FUNCTION "FC20 Motor 1O1I" : VOID	// FC 20
TITLE = Block for motor actuation and fault monitoring
//Erstellung:
//Datum        Bearbeiter                                                 Version
//--------------------------------------------------------------------------------
//26.06.97     H.Rüttling (rh)                                            01.00.00
//
//Änderungen:
//Nr. Datum    Bearb Änderung                                       Marke  Version
//--------------------------------------------------------------------------------
//01  09.02.99 sra   Einfügen der Handbedienuung                    ()    01.01.00
//02  16.04.99 sra   Fehlerbeseitigung Störungsquittierung          ()    01.01.01
//03  23.07.99 sra   Ausg. wird auch bei Simulation gesetzt         ()    01.01.02
//04  19.10.99 sra   "in" Reparaturschalter gelöscht                ()    01.02.00
//05  03.11.99 hus   Parameter eingefügt "FU in Betrieb"            ()    01.03.00
//06  18.09.00 sra   komplette Überarbeitung / neue Struktur        ()    02.00.00
//07  08.11.02 sra   Änderung Betriebsstundenzähler (zählt falsch)  (007) 02.01.00
//08  31.10.05 sra   Ansteuerung Handbedienung im Automode rücksetz.
//                   Handbedienung zentral sperren                  (008) 02.02.00
//09  04.09.06 sra   Änderung Störungsquittierung                   (009) 02.03.00
//10  20.11.07 gea   Handmode zurücksetzen wenn Handmode gesperrt   (010) 02.03.01
//11  18.02.09 kmj   Objektststatus für OP ergänzt                  (011) 02.04.00
//12  20.03.09 kal   Objektststatus für OP ergänzt (überarbeitet)   (012) 02.04.01
//13  05.12.13 sra   "Anlage ein" eingefügt (Not-Aus-Konzept)       (013) 02.05.00
//________________________________________________________________________________
//Funktion:
//
//-Der Baustein steuert den Ablauf eines Motors mit 1 Ausgang und 1 Eingang durch 
// setzten des Eingangsparameters "in_Ansteuerung_Motor".
//
//-Der Ausgang wird nur angesteuert wenn der Eingang "in_Anlage_ein" = true
// ist. Diese Funktion ist vorhanden, um bei einem Not-Halt die Anlage vor 
// unkontrolliertem Einschalten zu schützen. 
//
//-Ist in der Motorstruktur die Taktfunktion freigegeben wird bei Freigabe des 
// Motors der Ausgang entsprechend der Impuls-/Pausezeit angesteuert.
// !!Der Baustein arbeitet nur mit vollen Sekunden!!
//
//-Der Baustein überwacht den Zustand des Ausgangs und des Eingangs und generiert 
// nach Ablauf der "Sollzeit Störung" eine Störmeldung
//
//-Ist das Bit "Simulation" auf TRUE, so wird der Eingang simuliert.
//
//-Ist die Kennung "Betriebsstundenzähler_ein" aktiviert werden die Laufzeit 
// des Motors aufsummiert. Dies erfolgt mit setzen des Ausgangs.
//
//-Der Baustein kopiert die Parameter "in_Eingang_Motor", "io_Ausgang_Motor", 
// "in_Quitt_Stoerung" und "io_Stoerung" in die angegebene Datenstruktur zur 
// Visualisierung auf einem Farbgrafiksystem. Diese Parameter müssen folglich 
// nicht mehr extern umkopiert werden.
//
//-Ist der Parameter "in_Handbedienung_erlaubt" angewählt kann der Motor über 
// eine Farbgrafik oder ein Bedienterminal manuell angesteuert werden
//
AUTHOR : rh
FAMILY : AZO
VERSION : 0.0
VAR_INPUT
  in_Handbedienung_erlaubt : BOOL ;	//1 = manual operation permitted, 0 = manual operation not permitted/locked
  in_Quitt_Stoerung_noetig : BOOL ;	//1 = fault acknowledgement required, 0 = automatic fault acknowledgement
  in_Anlage_ein : BOOL ;	//Anlage bzw. Anlagenbereich nach Not-Halt freigegeben
  in_Quitt_Stoerung : BOOL ;	//Fault acknowledgement when fault_acknowledgement_required = 1
  in_Ansteuerung_Motor : BOOL ;	//Actuation of motor in automatic mode
  in_Eingang_Motor : BOOL ;	//Input of motor
END_VAR
VAR_IN_OUT
  io_Ausgang_Motor : BOOL ;	//Output of motor
  io_Motor_in_Betrieb : BOOL ;	//Signal "motor in operation"
  io_Stoerung : BOOL ;	//Signal "motor fault"
  io_Motorstruktur : ANY ;	//ANY pointer of motor structure
END_VAR
VAR_TEMP
  Freigabe_Takt : BOOL ;
  Start_mit_Impuls : BOOL ;
  Dauertakt : BOOL ;
  Taktausgang : BOOL ;
  Taktanzahl_erreicht : BOOL ;
  Diskrepanz : BOOL ;
  Impulszeit : REAL ;
  Pausezeit : REAL ;
  Sollanzahl_Takte : INT ;
  Zeitzaehler : REAL ;
  Taktzaehler : INT ;
  Objektstatus : INT ;
END_VAR
BEGIN
NETWORK
TITLE = Anfangs-DW der Struktur aus ANY-Zeiger auslesen
      L     P##io_Motorstruktur;
      LAR2;
      L     D [AR2,P#6.0];
      LAR2;
NETWORK
TITLE = Simulation
      AN    DIX [AR2,P#3.5];	// Simulation ein (Struktur)
      JC    ESIM;
      A     #io_Ausgang_Motor;
      =     #in_Eingang_Motor;
ESIM: NOP   0;
NETWORK
TITLE = Umschaltung Hand-/Automatikmode 
      A     DIX [AR2,P#2.7];	// Handmode von Farbgrafik (Struktur)
      AN    DIX [AR2,P#3.1];	// Handmode gesperrt (Struktur)
      AN    "M 0.0 Lock Man.Operation";	// Handbedienung zentral sperren (008)
      S     DIX [AR2,P#2.6];	// Handmode zu Farbgrafik (Struktur)
      ON    DIX [AR2,P#2.7];	// Handmode von Farbgrafik (Struktur)
      ON    #in_Handbedienung_erlaubt;
      O     "M 0.0 Lock Man.Operation";	// Handbedienung zentral sperren (008)
      O     DIX [AR2,P#3.1];	// Handmode gesperrt (Struktur)//(010)
      R     DIX [AR2,P#2.6];	// Handmode zu Farbgrafik (Struktur)
      R     DIX [AR2,P#2.7];	// Handmode zu Farbgrafik (Struktur) (008)
NETWORK
TITLE = Ansteuerung Handmode zurücksetzen
//(008) 
      AN    DIX [AR2,P#2.6];	// Handmode zu Farbgrafik (Struktur)
      R     DIX [AR2,P#3.0];	// Ansteuerung Handmode von Farbgrafik (Struktur)
NETWORK
TITLE = Daten für Takt in temporäre Variablen laden
      A     #in_Anlage_ein;	// (013)
      A     #in_Ansteuerung_Motor;
      A     DIX [AR2,P#3.6];	// Freigabe Takt (Struktur)
      =     #Freigabe_Takt;
      A     DIX [AR2,P#3.2];	// Start mit Impuls (Struktur)
      =     #Start_mit_Impuls;
      A     DIX [AR2,P#3.3];	// Taktanzahl erreicht (Struktur)
      =     #Taktanzahl_erreicht;
      A     DIX [AR2,P#3.4];	// Dauertakt (Struktur)
      =     #Dauertakt;
      A     DIX [AR2,P#3.7];	// Taktausgang (Struktur)
      =     #Taktausgang;
      L     DID [AR2,P#8.0];	// Impulszeit (Struktur)
      T     #Impulszeit;
      L     DID [AR2,P#12.0];	// Pausezeit (Struktur)
      T     #Pausezeit;
      L     DIW [AR2,P#20.0];	// Sollanzahl Takte (Struktur)
      T     #Sollanzahl_Takte;
      L     DID [AR2,P#16.0];	// Impuls-/Pausezähler (Struktur)
      T     #Zeitzaehler;
      L     DIW [AR2,P#22.0];	// Taktzähler (Struktur)
      T     #Taktzaehler;
NETWORK
TITLE = Takt generieren
      CALL  "FC2 Cycle Gen Timer Emul" (
           in_Freigabe              := #Freigabe_Takt,
           in_Rueckmeldung          := #in_Eingang_Motor,
           in_Start_mit_Impuls      := #Start_mit_Impuls,
           in_Dauertakt             := #Dauertakt,
           in_Impuls                := "M 4.5 Imp Cycle 1,0-sec",
           in_Impulszeit_in_100ms   := 10,
           in_Impulszeit            := #Impulszeit,
           in_Pausezeit             := #Pausezeit,
           in_Sollanzahl_Takte      := #Sollanzahl_Takte,
           io_Taktausgang           := #Taktausgang,
           io_Taktanzahl_erreicht   := #Taktanzahl_erreicht,
           io_Zeitzaehler           := #Zeitzaehler,
           io_Taktzaehler           := #Taktzaehler);
NETWORK
TITLE = Ansteuerung Ausgang des Motors
      A     #in_Anlage_ein;	// (013)
      AN    DIX [AR2,P#2.2];	// Motor gesperrt (Struktur)
      A(;
      AN    #in_Quitt_Stoerung_noetig;
      O;
      A     #in_Quitt_Stoerung_noetig;	// Wenn die Stoerung quittiert werden muß 
      AN    #io_Stoerung;	// wird der Ausgang bei einer anstehenden
      );	// Stoerung zurück gesetzt
      A(;
      AN    DIX [AR2,P#2.6];	// Automatikmode zu Farbgrafik (Struktur)
      AN    DIX [AR2,P#3.6];	// Freigabe Takt (Struktur)
      A     #in_Ansteuerung_Motor;
      O;
      AN    DIX [AR2,P#2.6];	// Automatikmode zu Farbgrafik (Struktur)
      A     DIX [AR2,P#3.6];	// Freigabe Takt (Struktur)
      A     #Taktausgang;
      O;
      A     DIX [AR2,P#2.6];	// Handmode zu Farbgrafik (Struktur)
      A     DIX [AR2,P#3.0];	// Ansteuerung Handmode von Farbgrafik (Struktur)
      );
      O;
      A     #in_Anlage_ein;	// (013)
      A     DIX [AR2,P#24.0];	// FU in Betrieb (Struktur)              
      A     #io_Ausgang_Motor;	// Ausschalten nur möglich, wenn Bit = 0 
      =     #io_Ausgang_Motor;
NETWORK
TITLE = Betriebsmeldung
      A     #io_Ausgang_Motor;
      A     #in_Eingang_Motor;
      =     #io_Motor_in_Betrieb;
NETWORK
TITLE = Diskrepanz feststellen
      A     #io_Ausgang_Motor;
      AN    #in_Eingang_Motor;
      O;
      A     #in_Eingang_Motor;
      AN    #io_Ausgang_Motor;
      =     #Diskrepanz;
NETWORK
TITLE = Störungszähler
      A     #in_Quitt_Stoerung_noetig;
      AN    #in_Quitt_Stoerung;
      A     #io_Stoerung;
      O;
      A     #Diskrepanz;
      AN    #in_Quitt_Stoerung;	// (009)
      O;	// (009)
      AN    #in_Quitt_Stoerung_noetig;	// (009)
      A     #Diskrepanz;	// (009)
      JC    SZ1;
      L     0;	// Wenn keine Diskrepanz dann Zähler löschen
      T     DIW [AR2,P#6.0];	// Istzeit Störung (Struktur)
      JU    ESZ;
// Störungszähler in jeder Sekunde erhöhen
SZ1:  O     #io_Stoerung;
      ON    "M 4.5 Imp Cycle 1,0-sec";	// Sekundenimpuls (Standardmerker)
      JC    ESZ;
      L     DIW [AR2,P#6.0];	// Istzeit Störung (Struktur)
      INC   1;
      T     DIW [AR2,P#6.0];	// Istzeit Störung (Struktur)
ESZ:  NOP   0;
NETWORK
TITLE = Störmeldung ausgeben
      L     DIW [AR2,P#6.0];	// Istzeit Störung (Struktur)
      L     DIW [AR2,P#4.0];	// Sollzeit Störung (Struktur)
      >=I;
      =     #io_Stoerung;
NETWORK
TITLE = Stoerung quittieren
      O     #Diskrepanz;	// Stoerung steht noch an
      ON    #io_Stoerung;
      JC    ESQ;
      ON    #in_Quitt_Stoerung_noetig;	// Stoerung muß quittiert werden ?
      JC    SQ1;	// Stoerung muß nicht quittiert werden
      A     #in_Quitt_Stoerung;
SQ1:  R     #io_Stoerung;
ESQ:  NOP   0;
NETWORK
TITLE = Betriebsstundenzähler
//jede Sekunde wird der Sekundenzähler erhöht und beim erreichen von 3600 
//Sekunden wird eine Betriebsstunde addiert. (nur über Gleitpunktwert zu ungenau)
      ON    DIX [AR2,P#0.3];	// Kennung Betriebsstundenzähler ein (Struktur)
      ON    #io_Ausgang_Motor;
      ON    "M 4.5 Imp Cycle 1,0-sec";	// Sekundentakt
      JC    EBSZ;
      L     DIW [AR2,P#44.0];	// Betriebsstunden Sekundenzähler bis 3600 (007)
      L     1;	// (007)
      +I;	// (007)
      T     DIW [AR2,P#44.0];	// Betriebsstunden Sekundenzähler bis 3600 (007)
      L     3600;	// (007)
      <I;	// (007)
      JC    EBSZ;	// (007)
      L     DID [AR2,P#32.0];	// Betriebsstundenzähler (007)
      L     1.000000e+00;	// (007)
      +R;	// (007)
      T     DID [AR2,P#32.0];	// Betriebsstundenzähler (007)
      L     0;	// (007)
      T     DIW [AR2,P#44.0];	// Betriebsstunden Sekundenzähler bis 3600 (007)
EBSZ: NOP   0;
NETWORK
TITLE = Betriebsstundenzähler zurücksetzten
      AN    DIX [AR2,P#30.0];	// Reset Betriebsstundenzähler (Struktur)
      JC    E_RB;
      L     0.000000e+00;
      T     DID [AR2,P#32.0];	// Betriebsstundenzähler (Struktur)
      CLR;
      =     DIX [AR2,P#30.0];	// Reset Betriebsstundenzähler (Struktur)
E_RB: NOP   0;
NETWORK
TITLE = Warnmeldung Betriebsstundenzähler erzeugen
      A(;
      L     DID [AR2,P#32.0];	// Betriebsstundenzähler (Struktur)
      L     DID [AR2,P#36.0];	// Sollzeit Warnung (Struktur)
      >R;
      );
      A(;
      L     DID [AR2,P#36.0];	// Sollzeit Warnung (Struktur)
      L     0.000000e+00;
      <>R;
      );
      =     DIX [AR2,P#30.1];	// Warnmeldung Betriebsstundenzähler (Struktur)
NETWORK
TITLE = Alarmmeldung Betriebsstundenzähler erzeugen
      A(;
      L     DID [AR2,P#32.0];	// Betriebsstundenzähler (Struktur)
      L     DID [AR2,P#40.0];	// Sollzeit Alarm (Struktur)
      >R;
      );
      A(;
      L     DID [AR2,P#40.0];	// Sollzeit Alarm (Struktur)
      L     0.000000e+00;
      <>R;
      );
      =     DIX [AR2,P#30.2];	// Warnmeldung Betriebsstundenzähler (Struktur)
NETWORK
TITLE = Objektstatus für Visualisation OP // (011)(012)
//Stati:
//-------
//1 = nicht in Betrieb, keine Störung ==> Farborschlag weiß
//5 = angesteuert, in Betrieb, keine Störung ==> Farbvorschalg grün
//9 = angesteuert, nicht in Betrieb, keine Störung ==> Farbvorschalg grau
//16 = Störung ==> Farbvorschalg rot
// 1 = nicht in Betrieb, keine Störung ==> Farborschlag weiß
      L     1;
      AN    #io_Ausgang_Motor;
      AN    #in_Eingang_Motor;
      AN    #io_Stoerung;
      JC    disp;
// 5 = angesteuert, in Betrieb, keine Störung ==> Farbvorschalg grün
      L     5;
      A     #io_Ausgang_Motor;
      A     #in_Eingang_Motor;
      AN    #io_Stoerung;
      JC    disp;
// 9 = angesteuert, nicht in Betrieb, keine Störung ==> Farbvorschalg grau
      L     9;
      A     #io_Ausgang_Motor;
      AN    #in_Eingang_Motor;
      AN    #io_Stoerung;
      JC    disp;
// 16 = Störung ==> Farbvorschalg rot
      L     16;
      A     #io_Stoerung;
      JC    disp;
      L     0;
disp: T     #Objektstatus;
NETWORK
TITLE = Daten in Struktur speichern
      A     #in_Anlage_ein;	// (013)
      =     DIX [AR2,P#46.0];	// (013) Anlage ein (Struktur)
      A     #in_Eingang_Motor;
      =     DIX [AR2,P#2.1];	// Eingang Motor (Struktur)
      A     #io_Ausgang_Motor;
      =     DIX [AR2,P#2.0];	// Ausgang Motor (Struktur)
      A     #io_Motor_in_Betrieb;
      =     DIX [AR2,P#2.4];	// Motor in Betrieb (Struktur)
      A     #io_Stoerung;
      =     DIX [AR2,P#2.5];	// Störung (Struktur)
      A     #Taktanzahl_erreicht;
      =     DIX [AR2,P#3.3];	// Taktanzahl erreicht (Struktur)
      A     #Taktausgang;
      =     DIX [AR2,P#3.7];	// Taktausgang (Struktur)
      L     #Zeitzaehler;
      T     DID [AR2,P#16.0];	// Impuls-/Pausezähler (Struktur)
      L     #Taktzaehler;
      T     DIW [AR2,P#22.0];	// Taktzähler (Struktur)
      L     #Objektstatus;	// (011)
      T     DIW [AR2,P#48.0];	// #Objektstatus  (Struktur)   // (011)
NETWORK
TITLE = ENDE
      NOP   0;
END_FUNCTION

FUNCTION "FC21 Valve 10-2I" : VOID	// FC 21
TITLE = Block for valve actuation and fault monitoring
//Erstellung:
//Datum        Bearbeiter                                                 Version
//--------------------------------------------------------------------------------
//26.06.97     H.Rüttling (rh)                                            01.00.00
//
//Änderungen:
//Nr. Datum    Bearb Änderung                                       Marke  Version
//--------------------------------------------------------------------------------
//01  09.02.99 sra   Einfügen der Handbedienuung                    ()    01.01.00
//02  16.04.99 sra   Fehlerbeseitigung Störungsquittierung          ()    01.01.01
//03  21.05.99 jm    Ventiltyp 0 eingefügt                          ()    01.02.00
//04  23.07.99 sra   Ausg. wird auch bei Simulation gesetzt         ()    01.02.01
//06  18.09.00 sra   komplette Überarbeitung / neue Struktur        ()    02.00.00
//07  31.10.05 sra   Ansteuerung Handbedienung im Automode rücksetz.
//                   Handbedienung zentral sperren                  (007) 02.01.00
//08  04.09.06 sra   Änderung Störungsquittierung                   (008) 02.02.00
//09  18.02.09 kmj   Objektststatus für OP ergänzt                  (009) 02.03.00
//10  20.03.09 kal   Objektststatus für OP ergänzt (überarbeitet)   (010) 02.03.01
//11  25.03.09 kal   1A0E-Objekt kann verzögert "in Betrieb" melden (011) 02.03.02
//12  25.03.09 kal   INC nach + geändert                            (012) 02.03.03
//13  20.11.07 gea   Handmode zurücksetzen wenn Handmode gesperrt   (013) 02.03.04
//14  14.07.09 kal   Objektstatus überarbeitet                      (014) 02.03.05
//15  05.12.13 sra   "Anlage ein" eingefügt (Not-Aus-Konzept)       (015) 02.04.00
//________________________________________________________________________________
//Funktion:
//
//-Der Parameter VENTIL_TYP unterscheidet zwischen 4 verschiedenen Ventiltypen
// Typ 0 = Ventil ohne Rückmeldung
// Typ 1 = Ventil oder Klappe mit der Rückmeldung angesteuert und nicht 
//        angesteuert: 1. Ausgang auf, Eingang auf, Eingang zu
//                     2. Ausgang zu , Eingang zu , Eingang auf
// TYP 2 = Ventil oder Klappe mit der Rückmeldung angesteuert
//                     1. Ausgang auf, Eingang auf
//                     2. Ausgang zu , Eingang zu 
// TYP 3 = Ventil oder Klappe mit der Rückmeldung nicht angesteuert
//                     1. Ausgang auf, Eingang zu
//                     2. Ausgang zu , Eingang auf 
//
//-Der Baustein steuert den Ablauf eines Ventils mit 1 Ausgang und 0-2 Eingängen
// durch setzten des Eingangsparameters "in_Ansteuerung_Ventil".
//
//-Der Ausgang wird nur angesteuert wenn der Eingang "in_Anlage_ein" = true
// ist. Diese Funktion ist vorhanden, um bei einem Not-Halt die Anlage vor 
// unkontrolliertem Einschalten zu schützen. 
//
//-Ist in der Ventilstruktur die Taktfunktion freigegeben wird bei Freigabe des 
// Ventils der Ausgang entsprechend der Impuls-/Pausezeit angesteuert.
//
//-Der Baustein überwacht den Zustand des Ausgangs und der Eingänge und generiert 
// nach Ablauf der "Sollzeit Störung" eine Störmeldung
//
//-Ist das Bit "Simulation" auf TRUE, so werden die Eingänge simuliert.
//
//-Ist die Kennung "Schalthäufigkeitszähler_ein" aktiviert werden die
// Ansteuerungen des Ventils aufsummiert. Dies erfolgt mit setzen des Ausgangs.
//
//-Der Baustein kopiert die Parameter "in_Eingang_...", "io_Ausgang_Ventil", 
// "in_Quitt_Stoerung" und "io_Stoerung" in die angegebene Datenstruktur zur 
// Visualisierung auf einem Farbgrafiksystem. Diese Parameter müssen folglich 
// nicht mehr extern umkopiert werden.
//
//-Ist der Parameter "in_Handbedienung_erlaubt" angewählt kann das Ventil über 
// eine Farbgrafik oder ein Bedienterminal manuell angesteuert werden
//
AUTHOR : rh
FAMILY : AZO
VERSION : 0.0
VAR_INPUT
  in_Ventil_Typ : INT ;	//see Functional description below
  in_Handbedienung_erlaubt : BOOL ;	//1 = manual operation permitted, 0 = manual operation not permitted/locked
  in_Quitt_Stoerung_noetig : BOOL ;	//1 = fault acknowledgement required, 0 = automatic fault acknowledgement
  in_Quitt_Stoerung : BOOL ;	//Fault acknowledgement when fault_acknowledgement_required = 1
  in_Anlage_ein : BOOL ;	//Anlage bzw. Anlagenbereich nach Not-Halt freigegeben
  in_Ansteuerung_Ventil : BOOL ;	//Actuation of valve in automatic mode
  in_Eingang_angesteuert : BOOL ;	//Valve intake when actuated
  in_Eingang_nicht_angest : BOOL ;	//Valve intake when not actuated
END_VAR
VAR_IN_OUT
  io_Ausgang_Ventil : BOOL ;	//Valve outlet
  io_Ventil_in_Betrieb : BOOL ;	//Signal "valve in operation" (actuated)
  io_Stoerung : BOOL ;	//Signal "valve fault"
  io_Ventilstruktur : ANY ;	//ANY pointer of valve structure
END_VAR
VAR_TEMP
  Freigabe_Takt : BOOL ;
  Rueckmeldung : BOOL ;
  Start_mit_Impuls : BOOL ;
  Dauertakt : BOOL ;
  Taktausgang : BOOL ;
  Taktanzahl_erreicht : BOOL ;
  Diskrepanz : BOOL ;
  positive_Flanke : BOOL ;
  Impulszeit : REAL ;
  Pausezeit : REAL ;
  Sollanzahl_Takte : INT ;
  Zeitzaehler : REAL ;
  Taktzaehler : INT ;
  Objektstatus : INT ;
END_VAR
BEGIN
NETWORK
TITLE = Anfangs-DW der Struktur aus ANY-Zeiger auslesen
      L     P##io_Ventilstruktur;
      LAR2;
      L     D [AR2,P#6.0];
      LAR2;
NETWORK
TITLE = Simulation
      AN    DIX [AR2,P#3.5];	// Simulation ein (Struktur)
      JC    ESIM;
      A     #io_Ausgang_Ventil;
      =     #in_Eingang_angesteuert;
      AN    #io_Ausgang_Ventil;
      =     #in_Eingang_nicht_angest;
      L     #in_Ventil_Typ;
      L     3;
      <>I;
      JC    ESIM;
      CLR;
      =     #in_Eingang_angesteuert;
      AN    #io_Ausgang_Ventil;
      =     #in_Eingang_nicht_angest;
ESIM: NOP   0;
NETWORK
TITLE = Umschaltung Hand-/Automatikmode 
      A     DIX [AR2,P#2.7];	// Handmode von Farbgrafik (Struktur)
      AN    DIX [AR2,P#3.1];	// Handmode gesperrt (Struktur)
      AN    "M 0.0 Lock Man.Operation";	// Handbedienung zentral sperren (007)
      S     DIX [AR2,P#2.6];	// Handmode zu Farbgrafik (Struktur)
      ON    DIX [AR2,P#2.7];	// Handmode von Farbgrafik (Struktur)
      ON    #in_Handbedienung_erlaubt;
      O     "M 0.0 Lock Man.Operation";	// Handbedienung zentral sperren (007)
      O     DIX [AR2,P#3.1];	// Handmode gesperrt (Struktur)//(013)
      R     DIX [AR2,P#2.6];	// Handmode zu Farbgrafik (Struktur)
      R     DIX [AR2,P#2.7];	// Handmode von Farbgrafik (Struktur) (007)
NETWORK
TITLE = Ansteuerung Handmode zurücksetzen
//(007) 
      AN    DIX [AR2,P#2.6];	// Handmode zu Farbgrafik (Struktur)
      R     DIX [AR2,P#3.0];	// Ansteuerung Handmode von Farbgrafik (Struktur)
NETWORK
TITLE = Daten für Takt in temporäre Variablen laden
      A     #in_Anlage_ein;	// (015)
      A     #in_Ansteuerung_Ventil;
      A     DIX [AR2,P#3.6];	// Freigabe Takt (Struktur)
      =     #Freigabe_Takt;
      A     DIX [AR2,P#3.2];	// Start mit Impuls (Struktur)
      =     #Start_mit_Impuls;
      A     DIX [AR2,P#3.3];	// Taktanzahl erreicht (Struktur)
      =     #Taktanzahl_erreicht;
      A     DIX [AR2,P#3.4];	// Dauertakt (Struktur)
      =     #Dauertakt;
      A     DIX [AR2,P#3.7];	// Taktausgang (Struktur)
      =     #Taktausgang;
      L     DID [AR2,P#8.0];	// Impulszeit (Struktur)
      T     #Impulszeit;
      L     DID [AR2,P#12.0];	// Pausezeit (Struktur)
      T     #Pausezeit;
      L     DID [AR2,P#16.0];	// Impuls-/Pausezähler (Struktur)
      T     #Zeitzaehler;
      L     DIW [AR2,P#20.0];	// Sollanzahl Takte (Struktur)
      T     #Sollanzahl_Takte;
      L     DIW [AR2,P#22.0];	// Taktzähler (Struktur)
      T     #Taktzaehler;
NETWORK
TITLE = Rückmeldung für Takt
      A(;
      L     #in_Ventil_Typ;
      L     0;
      ==I;
      );
      A     #io_Ausgang_Ventil;
      O;
      A(;
      L     #in_Ventil_Typ;
      L     1;
      ==I;
      );
      A     #in_Eingang_angesteuert;
      O;
      A(;
      L     #in_Ventil_Typ;
      L     2;
      ==I;
      );
      A     #in_Eingang_angesteuert;
      O;
      A(;
      L     #in_Ventil_Typ;
      L     3;
      ==I;
      );
      AN    #in_Eingang_nicht_angest;
      =     #Rueckmeldung;
NETWORK
TITLE = Takt generieren
      CALL  "FC2 Cycle Gen Timer Emul" (
           in_Freigabe              := #Freigabe_Takt,
           in_Rueckmeldung          := #Rueckmeldung,
           in_Start_mit_Impuls      := #Start_mit_Impuls,
           in_Dauertakt             := #Dauertakt,
           in_Impuls                := "M 1.7 Cycle Timer-FC",
           in_Impulszeit_in_100ms   := "MW 6 Timer Val Cycle FCs",
           in_Impulszeit            := #Impulszeit,
           in_Pausezeit             := #Pausezeit,
           in_Sollanzahl_Takte      := #Sollanzahl_Takte,
           io_Taktausgang           := #Taktausgang,
           io_Taktanzahl_erreicht   := #Taktanzahl_erreicht,
           io_Zeitzaehler           := #Zeitzaehler,
           io_Taktzaehler           := #Taktzaehler);
NETWORK
TITLE = Ansteuerung Ventil
      A     #in_Anlage_ein;	// (015)
      A(;
      ON    #in_Quitt_Stoerung_noetig;
      O;
      A     #in_Quitt_Stoerung_noetig;
      AN    #io_Stoerung;
      );
      A(;
      AN    DIX [AR2,P#2.6];	// Automatikmode zu Farbgrafik (Struktur)
      AN    DIX [AR2,P#3.6];	// Freigabe Takt (Struktur)
      A     #in_Ansteuerung_Ventil;
      O;
      AN    DIX [AR2,P#2.6];	// Automatikmode zu Farbgrafik (Struktur)
      A     DIX [AR2,P#3.6];	// Freigabe Takt (Struktur)
      A     #Taktausgang;
      O;
      A     DIX [AR2,P#2.6];	// Handmode zu Farbgrafik (Struktur)
      A     DIX [AR2,P#3.0];	// Ansteuerung Handmode von Farbgrafik (Struktur)
      );
      =     #io_Ausgang_Ventil;
NETWORK
TITLE = Ventiltyp festlegen
      L     #in_Ventil_Typ;
      L     0;
      ==I;
      JC    TYP0;	// Sprung zu Ventil Typ 0
      TAK;
      L     1;
      ==I;
      JC    TYP1;	// Sprung zu Ventil Typ 1
      TAK;
      L     2;
      ==I;
      JC    TYP2;	// Sprung zu Ventil Typ 2
      TAK;
      L     3;
      ==I;
      JC    TYP3;	// Sprung zu Ventil Typ 3
      JU    ENDE;
NETWORK
TITLE = Betriebsmeldung Typ 0 (kein Eingang)
TYP0: A     #io_Ausgang_Ventil;
      A(;	// (011)
      L     DIW [AR2,P#40.0];	// (011) Istzeit Verzögerung (Struktur) 
      L     DIW [AR2,P#38.0];	// (011) Sollzeit Verzögerung (Struktur)
      >=I;	// (011)
      );	// (011)
      =     #io_Ventil_in_Betrieb;	// Betriebsmeldung anzeigen
NETWORK
TITLE = Istzähler Verzögerung hochzählen (011)
      A     #io_Ausgang_Ventil;
      AN    "M 4.5 Imp Cycle 1,0-sec";	// Sekundenimpuls (Standardmerker)
      O     #io_Ventil_in_Betrieb;	// Betriebsmeldung anzeigen
      JC    KVZ;
      L     DIW [AR2,P#40.0];	// Istzeit Verzögerung (Struktur)
      +     1;
      T     DIW [AR2,P#40.0];	// Istzeit Verzögerung (Struktur)
KVZ:  NOP   0;
NETWORK
TITLE = Istzähler Verzögerung zurücksetzen (011)
      O     #io_Ausgang_Ventil;
      JC    RVZ;
      L     0;
      T     DIW [AR2,P#40.0];	// Istzeit Verzögerung (Struktur)
RVZ:  NOP   0;
NETWORK
TITLE = Diskrepanz Typ 0 (kein Eingang)
      CLR;	// keine Diskrepanz möglich
      =     #Diskrepanz;
      JU    STOE;
NETWORK
TITLE = Betriebsmeldung Typ1 (Eingang angesteuert und nicht angesteuert)
TYP1: A     #io_Ausgang_Ventil;
      A     #in_Eingang_angesteuert;
      AN    #in_Eingang_nicht_angest;
      =     #io_Ventil_in_Betrieb;
NETWORK
TITLE = Diskrepanz Typ 1 (Eingang angesteuert und nicht angesteuert)
      A     #io_Ausgang_Ventil;
      AN    #in_Eingang_angesteuert;
      O;
      AN    #io_Ausgang_Ventil;
      AN    #in_Eingang_nicht_angest;
      O;
      A     #in_Eingang_angesteuert;
      A     #in_Eingang_nicht_angest;
      O;
      AN    #in_Eingang_angesteuert;
      AN    #in_Eingang_nicht_angest;
      =     #Diskrepanz;
      JU    STOE;
NETWORK
TITLE = Betriebsmeldung Typ 2 (Eingang angesteuert)
TYP2: A     #io_Ausgang_Ventil;
      A     #in_Eingang_angesteuert;
      =     #io_Ventil_in_Betrieb;
NETWORK
TITLE = Diskrepanz Typ 2 (Eingang angesteuert)
      A     #io_Ausgang_Ventil;
      AN    #in_Eingang_angesteuert;
      O;
      AN    #io_Ausgang_Ventil;
      A     #in_Eingang_angesteuert;
      =     #Diskrepanz;
      JU    STOE;
NETWORK
TITLE = Betriebsmeldung Typ 3 (Eingang nicht angesteuert)
TYP3: A     #io_Ausgang_Ventil;
      AN    #in_Eingang_nicht_angest;
      =     #io_Ventil_in_Betrieb;
NETWORK
TITLE = Diskrepanz Typ 3 (Eingang nicht angesteuert)
      A     #io_Ausgang_Ventil;
      A     #in_Eingang_nicht_angest;
      O;
      AN    #io_Ausgang_Ventil;
      AN    #in_Eingang_nicht_angest;
      =     #Diskrepanz;
NETWORK
TITLE = Störungszähler
STOE: A     #in_Quitt_Stoerung_noetig;
      AN    #in_Quitt_Stoerung;
      A     #io_Stoerung;
      O;
      A     #Diskrepanz;
      AN    #in_Quitt_Stoerung;	// (008)
      O;	// (008)
      AN    #in_Quitt_Stoerung_noetig;	// (008)
      A     #Diskrepanz;	// (008)
      JC    SZ1;
      L     0;	// Wenn keine Diskrepanz dann Zähler löschen
      T     DIW [AR2,P#6.0];	// Istzeit Störung (Struktur)
      JU    ESZ;
// Störungszähler in jeder Sekunde erhöhen
SZ1:  O     #io_Stoerung;
      ON    "M 4.5 Imp Cycle 1,0-sec";	// Sekundenimpuls (Standardmerker)
      JC    ESZ;
      L     DIW [AR2,P#6.0];	// Istzeit Störung (Struktur)
      +     1;	// (012)
      T     DIW [AR2,P#6.0];	// Istzeit Störung (Struktur)
ESZ:  NOP   0;
NETWORK
TITLE = Störmeldung ausgeben
      L     DIW [AR2,P#6.0];	// Istzeit Störung (Struktur)
      L     DIW [AR2,P#4.0];	// Sollzeit Störung (Struktur)
      >=I;
      =     #io_Stoerung;
NETWORK
TITLE = Stoerung quittieren
      O     #Diskrepanz;	// Stoerung steht noch an
      ON    #io_Stoerung;
      JC    ESQ;
      ON    #in_Quitt_Stoerung_noetig;	// Stoerung muß quittiert werden ?
      JC    SQ1;	// Stoerung muß nicht quittiert werden
      A     #in_Quitt_Stoerung;
SQ1:  R     #io_Stoerung;
ESQ:  NOP   0;
NETWORK
TITLE = Flankenauswertung Ausgang Ventil für Schalthäufigkeitzähler
      A     #io_Ausgang_Ventil;
      FP    DIX [AR2,P#24.3];	// Flankenmerker Ausgang (Struktur)
      =     #positive_Flanke;
NETWORK
TITLE = Schalthäufigkeitzähler
      ON    DIX [AR2,P#0.3];	// Kennung Schalthäufigkeitzähler ein (Struktur)
      ON    #positive_Flanke;
      JC    ESHZ;
      L     1.000000e+00;
      L     DID [AR2,P#26.0];	// Schalthäufigkeitzähler (Struktur)
      +R;
      T     DID [AR2,P#26.0];	// Schalthäufigkeitzähler (Struktur)
ESHZ: NOP   0;
NETWORK
TITLE = Schalthäufigkeitzähler zurücksetzten
      AN    DIX [AR2,P#24.0];	// Reset Schalthäufigkeitzähler (Struktur)
      JC    E_RS;
      L     0.000000e+00;
      T     DID [AR2,P#26.0];	// Schalthäufigkeitzähler (Struktur)
      CLR;
      =     DIX [AR2,P#24.0];	// Reset Schalthäufigkeitzähler (Struktur)
E_RS: NOP   0;
NETWORK
TITLE = Warnmeldung Schalthäufigkeitszähler erzeugen
      A(;
      L     DID [AR2,P#26.0];	// Schalthäufigkeitzähler (Struktur)
      L     DID [AR2,P#30.0];	// Sollwert Warnung (Struktur)
      >R;
      );
      A(;
      L     DID [AR2,P#30.0];	// Sollwert Warnung (Struktur)
      L     0.000000e+00;
      <>R;
      );
      =     DIX [AR2,P#24.1];	// Warnmeldung Schalthäufigkeitzähler (Struktur)
NETWORK
TITLE = Alarmmeldung Schalthäufigkeitszähler erzeugen
      A(;
      L     DID [AR2,P#26.0];	// Schalthäufigkeitzähler (Struktur)
      L     DID [AR2,P#34.0];	// Sollwert Alarm (Struktur)
      >R;
      );
      A(;
      L     DID [AR2,P#34.0];	// Sollwert Alarm (Struktur)
      L     0.000000e+00;
      <>R;
      );
      =     DIX [AR2,P#24.2];	// Alarmmeldung Schalthäufigkeitzähler (Struktur)
NETWORK
TITLE = Objektstatus für Visualisation OP (009) (010)
//Stati:
//-------
//1 = nicht in Betrieb, keine Störung ==> Farbvorschlag weiß
//5 = angesteuert, in Betrieb, keine Störung ==> Farbvorschlag grün
//9 = angesteuert, nicht in Betrieb, keine Störung ==> Farbvorschlag grau
//16 = Störung ==> Farbvorschlag rot
// 1 = nicht in Betrieb, keine Störung ==> Farbvorschlag weiß
      L     1;
      AN    #io_Ausgang_Ventil;
      AN    #io_Stoerung;
      AN    DIX [AR2,P#1.3];	// (014) Kennung "invers"
      O;
      A     #io_Ausgang_Ventil;
      A     #io_Ventil_in_Betrieb;
      AN    #io_Stoerung;
      A     DIX [AR2,P#1.3];	// (014) Kennung "invers"
      JC    disp;
// 5 = angesteuert, in Betrieb, keine Störung ==> Farbvorschlag grün
      L     5;
      A     #io_Ausgang_Ventil;
      A     #io_Ventil_in_Betrieb;
      AN    #io_Stoerung;
      AN    DIX [AR2,P#1.3];	// (014) Kennung "invers"
      O;
      AN    #io_Ausgang_Ventil;
      AN    #io_Stoerung;
      A     DIX [AR2,P#1.3];	// (014) Kennung "invers"
      JC    disp;
// 9 = angesteuert, nicht in Betrieb, keine Störung ==> Farbvorschlag grau
      L     9;
      A     #io_Ausgang_Ventil;
      AN    #io_Ventil_in_Betrieb;
      AN    #io_Stoerung;
      JC    disp;
// 16 = Störung ==> Farbvorschlag rot
      L     16;
      A     #io_Stoerung;
      JC    disp;
      L     0;
disp: T     #Objektstatus;
NETWORK
TITLE = Daten in Struktur speichern
      A     #in_Anlage_ein;	// (015)
      =     DIX [AR2,P#42.0];	// (015) Anlage ein (Struktur)
      A     #in_Eingang_angesteuert;
      =     DIX [AR2,P#2.1];	// Eingang angesteuert (Struktur)
      A     #in_Eingang_nicht_angest;
      =     DIX [AR2,P#2.2];	// Eingang nicht angesteuert (Struktur)
      A     #io_Ausgang_Ventil;
      =     DIX [AR2,P#2.0];	// Ausgang Ventil (Struktur)
      A     #io_Ventil_in_Betrieb;
      =     DIX [AR2,P#2.4];	// Ventil in Betrieb (Struktur)
      A     #io_Stoerung;
      =     DIX [AR2,P#2.5];	// Störung (Struktur)
      A     #Taktanzahl_erreicht;
      =     DIX [AR2,P#3.3];	// Taktanzahl erreicht (Struktur)
      A     #Taktausgang;
      =     DIX [AR2,P#3.7];	// Taktausgang (Struktur)
      L     #Zeitzaehler;
      T     DID [AR2,P#16.0];	// Impuls-/Pausezähler (Struktur)
      L     #Taktzaehler;
      T     DIW [AR2,P#22.0];	// Taktzähler (Struktur)
      L     #Objektstatus;	// (009)
      T     DIW [AR2,P#48.0];	// #Objektstatus  (Struktur)   // (009)
NETWORK
TITLE = ENDE
ENDE: NOP   0;
END_FUNCTION

FUNCTION "FC23 Valve 1-10O" : VOID	// FC 23
TITLE = Bock for actuating several cycled valves
//Erstellung:
//Datum       Bearbeiter                                                   Version
//--------------------------------------------------------------------------------
//14.06.99    A.Kirchgessner(kia)                                         01.00.00
//
//Änderungen:
//Nr. Datum    Bearb Änderung                                       Marke  Version
//--------------------------------------------------------------------------------
//01  16.07.99 kia   Fehlerbeseitigung                                    01.00.01
//02  12.08.99 sra   Fehlerbeseitigung mit Parameteränderung              01.01.00
//03  19.10.99 sra   Anpassung an neue Struktur                           01.02.00
//04  10.07.00 sra   Fehlerbeseitigung Taktgenerierung                    01.02.01
//05  10.07.00 sra   Änderung in Eingangsparameter                        01.03.00
//06  19.09.00 sra   komplette Überarbeitung / neue Struktur              02.00.00
//07  18.01.01 gea   Erweiterung auf 10 Ventile / neue Struktur           02.01.00
//08  27.03.02 sra   Meldung "Ventil in Betrieb" auch im Handmode   (008) 02.01.01
//09  04.02.03 kal   Fehlerbeseitigung Dauertakt                    (009) 02.01.02
//10  31.10.05 sra   Ansteuerung Handbedienung im Automode rücksetz.
//                   Handbedienung zentral sperren                  (010) 02.02.00
//11  18.02.09 kmj   Objektststatus für OP ergänzt                  (011) 02.03.00
//12  20.03.09 kal   Objektststatus für OP ergänzt (überarbeitet)   (012) 02.03.01
//13  24.04.09 gea   Handmode zurücksetzen wenn Handmode gesperrt   (013) 02.03.02
//14  05.12.13 sra   "Anlage ein" eingefügt (Not-Aus-Konzept)       (014) 02.04.00
//15  14.11.14 bhl   Anzeige "#io_Ventil_in_Betrieb" im Handmode    (015) 02.04.01
//16  11.08.15 sra   "#io_Ventil_in_Betrieb" nur wenn "Anlage ein"  (016) 02.04.02
//________________________________________________________________________________
//Eingesetzte Bausteine:
//
//FC2 : Version 01.01.XX
//________________________________________________________________________________
//Funktion:
//
//Der Baustein taktet die einzelnen Ventile der Reihe nach durch (Anzahl der 
//Ventile max. 10 Stück). 
//
//Die Ausgänge werden nur angesteuert wenn der Eingang "in_Anlage_ein" = true
//ist. Diese Funktion ist vorhanden, um bei einem Not-Halt die Anlage vor 
//unkontrolliertem Einschalten zu schützen. 
//
//Im Handmode werden die ausgewählten Ventile dauerhaft angesteuert. 
//
AUTHOR : kia
FAMILY : AZO
VERSION : 0.0
VAR_INPUT
  in_Handbedienung_erlaubt : BOOL ;	//1 = manual operation permitted, 0 = manual operation not permitted/locked
  in_Anlage_ein : BOOL ;	//Anlage bzw. Anlagenbereich nach Not-Halt freigegeben
  in_Ansteuerung_Ventil_T1 : BOOL ;	//Actuation of valve position 1 in automatic mode with cycle 1
  in_Ansteuerung_Ventil_T2 : BOOL ;	//Actuation of valve position 1 in automatic mode with cycle 2
END_VAR
VAR_IN_OUT
  io_Ausgang_Ventil_1 : BOOL ;	//Output 1. Valve
  io_Ausgang_Ventil_2 : BOOL ;	//Output 2. Valve
  io_Ausgang_Ventil_3 : BOOL ;	//Output 3. Valve
  io_Ausgang_Ventil_4 : BOOL ;	//Output 4. Valve
  io_Ausgang_Ventil_5 : BOOL ;	//Output 5. Valve
  io_Ausgang_Ventil_6 : BOOL ;	//Output 6. Valve
  io_Ausgang_Ventil_7 : BOOL ;	//Output 7. Valve
  io_Ausgang_Ventil_8 : BOOL ;	//Output 8. Valve
  io_Ausgang_Ventil_9 : BOOL ;	//Output 9. Valve
  io_Ausgang_Ventil_10 : BOOL ;	//Output 10. Valve
  io_Ventil_in_Betrieb : BOOL ;	//Signal "valve in operation" (actuated)
  io_Ventilstruktur : ANY ;	//ANY pointer of valve structure
END_VAR
VAR_TEMP
  Ventilansteuerung : BOOL ;	//Freigabe ein Ventil anzusteuern
  Freigabe_Takt : BOOL ;	//Cycle enable
  Rueckmeldung : BOOL ;	//wenn eines der Ventil agesteuert ist --> 1-Signal
  Start_mit_Impuls : BOOL ;
  Taktanzahl_erreicht : BOOL ;
  Dauertakt : BOOL ;	//Continuous cycle
  positive_Flanke : BOOL ;
  Hilfs_Anzahl_Takte : INT ;	//Sollvorgabe für FC2
  Aktuelles_Ventil : INT ;	//aktuelles Ventil
  Hilfswort_1 : INT ;
  Impulszeit_Takt : REAL ;
  Pausezeit_Takt : REAL ;
  Zeitzaehler : REAL ;
  Taktzaehler : INT ;
  Objektstatus : INT ;
END_VAR
BEGIN
NETWORK
TITLE = Anfangs-DW der Struktur aus ANY-Zeiger auslesen
      L     P##io_Ventilstruktur;
      LAR2;
      L     D [AR2,P#6.0];
      LAR2;	//Pointer auf Structuranfang
NETWORK
TITLE = Umschaltung Hand-/Automatikmode 
      A     DIX [AR2,P#3.6];	// Handmode von Farbgrafik (Struktur)
      AN    DIX [AR2,P#5.1];	// Handmode gesperrt (Struktur)
      AN    "M 0.0 Lock Man.Operation";	// Handbedienung zentral sperren (010)
      S     DIX [AR2,P#3.5];	// Handmode zu Farbgrafik (Struktur)
      ON    DIX [AR2,P#3.6];	// Handmode von Farbgrafik (Struktur)
      ON    #in_Handbedienung_erlaubt;
      O     "M 0.0 Lock Man.Operation";	// Handbedienung zentral sperren (010)
      O     DIX [AR2,P#5.1];	// Handmode gesperrt (Struktur) (013)
      R     DIX [AR2,P#3.5];	// Handmode zu Farbgrafik (Struktur)
      R     DIX [AR2,P#3.6];	// Handmode von Farbgrafik (Struktur) (010)
NETWORK
TITLE = Ansteuerung Handmode zurücksetzen
//(010) 
      AN    DIX [AR2,P#3.5];	// Handmode zu Farbgrafik (Struktur)
      R     DIX [AR2,P#3.7];	// Ansteuerung des 1. Ventils im Handmode von Farbgrafik (Struktur)
      R     DIX [AR2,P#4.0];	// Ansteuerung des 2. Ventils im Handmode von Farbgrafik (Struktur)
      R     DIX [AR2,P#4.1];	// Ansteuerung des 3. Ventils im Handmode von Farbgrafik (Struktur)
      R     DIX [AR2,P#4.2];	// Ansteuerung des 4. Ventils im Handmode von Farbgrafik (Struktur)
      R     DIX [AR2,P#4.3];	// Ansteuerung des 5. Ventils im Handmode von Farbgrafik (Struktur)
      R     DIX [AR2,P#4.4];	// Ansteuerung des 6. Ventils im Handmode von Farbgrafik (Struktur)
      R     DIX [AR2,P#4.5];	// Ansteuerung des 7. Ventils im Handmode von Farbgrafik (Struktur)
      R     DIX [AR2,P#4.6];	// Ansteuerung des 8. Ventils im Handmode von Farbgrafik (Struktur)
      R     DIX [AR2,P#4.7];	// Ansteuerung des 9. Ventils im Handmode von Farbgrafik (Struktur)
      R     DIX [AR2,P#5.0];	// Ansteuerung des 10. Ventils im Handmode von Farbgrafik (Struktur)
NETWORK
TITLE = Rueckmeldung Ventile + Ventilansteuerung
      O     #io_Ausgang_Ventil_1;
      O     #io_Ausgang_Ventil_2;
      O     #io_Ausgang_Ventil_3;
      O     #io_Ausgang_Ventil_4;
      O     #io_Ausgang_Ventil_5;
      O     #io_Ausgang_Ventil_6;
      O     #io_Ausgang_Ventil_7;
      O     #io_Ausgang_Ventil_8;
      O     #io_Ausgang_Ventil_9;
      O     #io_Ausgang_Ventil_10;
      =     #Rueckmeldung;
      =     #Ventilansteuerung;
NETWORK
TITLE = Daten für Takt in temporäre Variablen laden
//(009) komplettes Netzwerk gelöscht.
//Dauertakt nur, wenn Bit in Struktur = TRUE 
//Anzahl Takte ist egal!!!
      A     DIX [AR2,P#5.2];	// Start mit Impuls (Struktur)
      =     #Start_mit_Impuls;
      A     DIX [AR2,P#5.3];	// Taktanzahl erreicht (Struktur)
      =     #Taktanzahl_erreicht;
      A     DIX [AR2,P#5.4];	// Dauertakt (Struktur)
      =     #Dauertakt;
      L     DID [AR2,P#22.0];	// Impuls-/Pausezähler (Struktur)
      T     #Zeitzaehler;
      L     DIW [AR2,P#28.0];	// Taktzähler (Struktur)
      T     #Taktzaehler;
NETWORK
TITLE = Sollanzahl Takte
      AN    #Dauertakt;
      JC    ST_1;
      L     DIW [AR2,P#30.0];	// Anzahl Ventile (Struktur)
      T     #Hilfs_Anzahl_Takte;
ST_1: NOP   0;
      A     #Dauertakt;
      JC    ST_2;
      L     DIW [AR2,P#26.0];	// Sollanzahl Takte (Struktur)
      T     #Hilfs_Anzahl_Takte;
ST_2: NOP   0;
NETWORK
TITLE = Freigabe Takt
      A     #in_Anlage_ein;	// (014)
      A(;	// (014)
      O     #in_Ansteuerung_Ventil_T1;
      O     #in_Ansteuerung_Ventil_T2;
      );	// (014)
      =     #Freigabe_Takt;
NETWORK
TITLE = Takt umkopieren
      L     DID [AR2,P#6.0];	// Impulszeit Befüllung (Struktur)
      T     #Impulszeit_Takt;
      L     DID [AR2,P#10.0];	// Pausezeit Befüllung (Struktur)
      T     #Pausezeit_Takt;
      A     #in_Ansteuerung_Ventil_T1;
      JC    E_Tk;
      L     DID [AR2,P#14.0];	// Impulszeit Entleerung (Struktur)
      T     #Impulszeit_Takt;
      L     DID [AR2,P#18.0];	// Pausezeit Entleerung (Struktur)
      T     #Pausezeit_Takt;
E_Tk: NOP   0;
NETWORK
TITLE = Takt generieren
      CALL  "FC2 Cycle Gen Timer Emul" (
           in_Freigabe              := #Freigabe_Takt,
           in_Rueckmeldung          := #Rueckmeldung,
           in_Start_mit_Impuls      := #Start_mit_Impuls,
           in_Dauertakt             := #Dauertakt,
           in_Impuls                := "M 1.7 Cycle Timer-FC",
           in_Impulszeit_in_100ms   := "MW 6 Timer Val Cycle FCs",
           in_Impulszeit            := #Impulszeit_Takt,
           in_Pausezeit             := #Pausezeit_Takt,
           in_Sollanzahl_Takte      := #Hilfs_Anzahl_Takte,
           io_Taktausgang           := #Ventilansteuerung,
           io_Taktanzahl_erreicht   := #Taktanzahl_erreicht,
           io_Zeitzaehler           := #Zeitzaehler,
           io_Taktzaehler           := #Taktzaehler);
NETWORK
TITLE = aktuelles Ventil
      L     #Taktzaehler;
      L     DIW [AR2,P#30.0];	// Anzahl Ventile (Struktur)
      /I;
      T     #Hilfswort_1;
      L     #Hilfswort_1;
      L     DIW [AR2,P#30.0];	// Anzahl Ventile (Struktur)
      *I;
      L     -1;
      *I;
      L     #Taktzaehler;
      +I;
      L     1;
      +I;
      T     #Aktuelles_Ventil;
NETWORK
TITLE = aktuelles Ventil prüfen
      A(;
      L     #Aktuelles_Ventil;
      L     1;
      >=I;
      );
      A(;
      L     #Aktuelles_Ventil;
      L     DIW [AR2,P#30.0];	// Anzahl Ventile (Struktur)
      <=I;
      );
      JC    M1;
      L     1;
      T     #Aktuelles_Ventil;
M1:   NOP   0;
NETWORK
TITLE = Ansteuerung Ventil 1
      A     #in_Anlage_ein;	// (014)
      A(;	// (014)
      A(;
      L     #Aktuelles_Ventil;
      L     1;
      ==I;
      );
      A(;	// Automatikmode
      AN    DIX [AR2,P#3.5];	// Handmode zu Farbgrafik (Struktur)
      A     #Ventilansteuerung;
      AN    #Taktanzahl_erreicht;
      );
      O;	// Handmode 
      A     DIX [AR2,P#3.5];	// Handmode zu Farbgrafik (Struktur)
      A     DIX [AR2,P#3.7];	// Ansteuerung des 1. Ventils im Handmode von Farbgrafik (Struktur)
      );	// (014)
      =     #io_Ausgang_Ventil_1;
NETWORK
TITLE = Ansteuerung Ventil 2
      A     #in_Anlage_ein;	// (014)
      A(;	// (014)
      A(;
      L     #Aktuelles_Ventil;
      L     2;
      ==I;
      );
      A(;	// Automatikmode
      AN    DIX [AR2,P#3.5];	// Handmode zu Farbgrafik (Struktur)
      A     #Ventilansteuerung;
      AN    #Taktanzahl_erreicht;
      );
      O;	// Handmode 
      A     DIX [AR2,P#3.5];	// Handmode zu Farbgrafik (Struktur)
      A     DIX [AR2,P#4.0];	// Ansteuerung des 2. Ventils im Handmode von Farbgrafik (Struktur)
      );	// (014)
      =     #io_Ausgang_Ventil_2;
NETWORK
TITLE = Ansteuerung Ventil 3
      A     #in_Anlage_ein;	// (014)
      A(;	// (014)
      A(;
      L     #Aktuelles_Ventil;
      L     3;
      ==I;
      );
      A(;	// Automatikmode
      AN    DIX [AR2,P#3.5];	// Handmode zu Farbgrafik (Struktur)
      A     #Ventilansteuerung;
      AN    #Taktanzahl_erreicht;
      );
      O;	// Handmode 
      A     DIX [AR2,P#3.5];	// Handmode zu Farbgrafik (Struktur)
      A     DIX [AR2,P#4.1];	// Ansteuerung des 3. Ventils im Handmode von Farbgrafik (Struktur)
      );	// (014)
      =     #io_Ausgang_Ventil_3;
NETWORK
TITLE = Ansteuerung Ventil 4
      A     #in_Anlage_ein;	// (014)
      A(;	// (014)
      A(;
      L     #Aktuelles_Ventil;
      L     4;
      ==I;
      );
      A(;	// Automatikmode
      AN    DIX [AR2,P#3.5];	// Handmode zu Farbgrafik (Struktur)
      A     #Ventilansteuerung;
      AN    #Taktanzahl_erreicht;
      );
      O;	// Handmode 
      A     DIX [AR2,P#3.5];	// Handmode zu Farbgrafik (Struktur)
      A     DIX [AR2,P#4.2];	// Ansteuerung des 4. Ventils im Handmode von Farbgrafik (Struktur)
      );	// (014)
      =     #io_Ausgang_Ventil_4;
NETWORK
TITLE = Ansteuerung Ventil 5
      A     #in_Anlage_ein;	// (014)
      A(;	// (014)
      A(;
      L     #Aktuelles_Ventil;
      L     5;
      ==I;
      );
      A(;	// Automatikmode
      AN    DIX [AR2,P#3.5];	// Handmode zu Farbgrafik (Struktur)
      A     #Ventilansteuerung;
      AN    #Taktanzahl_erreicht;
      );
      O;	// Handmode 
      A     DIX [AR2,P#3.5];	// Handmode zu Farbgrafik (Struktur)
      A     DIX [AR2,P#4.3];	// Ansteuerung des 5. Ventils im Handmode von Farbgrafik (Struktur)
      );	// (014)
      =     #io_Ausgang_Ventil_5;
NETWORK
TITLE = Ansteuerung Ventil 6
      A     #in_Anlage_ein;	// (014)
      A(;	// (014)
      A(;
      L     #Aktuelles_Ventil;
      L     6;
      ==I;
      );
      A(;	// Automatikmode
      AN    DIX [AR2,P#3.5];	// Handmode zu Farbgrafik (Struktur)
      A     #Ventilansteuerung;
      AN    #Taktanzahl_erreicht;
      );
      O;	// Handmode 
      A     DIX [AR2,P#3.5];	// Handmode zu Farbgrafik (Struktur)
      A     DIX [AR2,P#4.4];	// Ansteuerung des 6. Ventils im Handmode von Farbgrafik (Struktur)
      );	// (014)
      =     #io_Ausgang_Ventil_6;
NETWORK
TITLE = Ansteuerung Ventil 7
      A     #in_Anlage_ein;	// (014)
      A(;	// (014)
      A(;
      L     #Aktuelles_Ventil;
      L     7;
      ==I;
      );
      A(;	// Automatikmode
      AN    DIX [AR2,P#3.5];	// Handmode zu Farbgrafik (Struktur)
      A     #Ventilansteuerung;
      AN    #Taktanzahl_erreicht;
      );
      O;	// Handmode 
      A     DIX [AR2,P#3.5];	// Handmode zu Farbgrafik (Struktur)
      A     DIX [AR2,P#4.5];	// Ansteuerung des 7. Ventils im Handmode von Farbgrafik (Struktur)
      );	// (014)
      =     #io_Ausgang_Ventil_7;
NETWORK
TITLE = Ansteuerung Ventil 8
      A     #in_Anlage_ein;	// (014)
      A(;	// (014)
      A(;
      L     #Aktuelles_Ventil;
      L     8;
      ==I;
      );
      A(;	// Automatikmode
      AN    DIX [AR2,P#3.5];	// Handmode zu Farbgrafik (Struktur)
      A     #Ventilansteuerung;
      AN    #Taktanzahl_erreicht;
      );
      O;	// Handmode 
      A     DIX [AR2,P#3.5];	// Handmode zu Farbgrafik (Struktur)
      A     DIX [AR2,P#4.6];	// Ansteuerung des 8. Ventils im Handmode von Farbgrafik (Struktur)
      );	// (014)
      =     #io_Ausgang_Ventil_8;
NETWORK
TITLE = Ansteuerung Ventil 9
      A     #in_Anlage_ein;	// (014)
      A(;	// (014)
      A(;
      L     #Aktuelles_Ventil;
      L     9;
      ==I;
      );
      A(;	// Automatikmode
      AN    DIX [AR2,P#3.5];	// Handmode zu Farbgrafik (Struktur)
      A     #Ventilansteuerung;
      AN    #Taktanzahl_erreicht;
      );
      O;	// Handmode 
      A     DIX [AR2,P#3.5];	// Handmode zu Farbgrafik (Struktur)
      A     DIX [AR2,P#4.7];	// Ansteuerung des 9. Ventils im Handmode von Farbgrafik (Struktur)
      );	// (014)
      =     #io_Ausgang_Ventil_9;
NETWORK
TITLE = Ansteuerung Ventil 10
      A     #in_Anlage_ein;	// (014)
      A(;	// (014)
      A(;
      L     #Aktuelles_Ventil;
      L     10;
      ==I;
      );
      A(;	// Automatikmode
      AN    DIX [AR2,P#3.5];	// Handmode zu Farbgrafik (Struktur)
      A     #Ventilansteuerung;
      AN    #Taktanzahl_erreicht;
      );
      O;	// Handmode 
      A     DIX [AR2,P#3.5];	// Handmode zu Farbgrafik (Struktur)
      A     DIX [AR2,P#5.0];	// Ansteuerung des 10. Ventils im Handmode von Farbgrafik (Struktur)
      );	// (014)
      =     #io_Ausgang_Ventil_10;
NETWORK
TITLE = Ausgang Betrieb
      AN    DIX [AR2,P#3.5];	// (015) Handmode zu Farbgrafik (Struktur)
      A     #in_Anlage_ein;	// (016)
      A(;
      O     #in_Ansteuerung_Ventil_T1;
      O     #in_Ansteuerung_Ventil_T2;	// (008)
      );
      A     #Dauertakt;
      O;
      AN    DIX [AR2,P#3.5];	// (015) Handmode zu Farbgrafik (Struktur)
      A     #in_Anlage_ein;	// (016)
      A(;
      O     #in_Ansteuerung_Ventil_T1;
      O     #in_Ansteuerung_Ventil_T2;
      );
      AN    #Dauertakt;
      AN    #Taktanzahl_erreicht;
      O;
      A     DIX [AR2,P#3.5];	// Handmode zu Farbgrafik (Struktur)
      A     #in_Anlage_ein;	// (016)
      A(;
      O     #io_Ausgang_Ventil_1;	// (008)
      O     #io_Ausgang_Ventil_2;	// (008)
      O     #io_Ausgang_Ventil_3;	// (008)
      O     #io_Ausgang_Ventil_4;	// (008)
      O     #io_Ausgang_Ventil_5;	// (008)
      O     #io_Ausgang_Ventil_6;	// (008)
      O     #io_Ausgang_Ventil_7;	// (008)
      O     #io_Ausgang_Ventil_8;	// (008)
      O     #io_Ausgang_Ventil_9;	// (008)
      O     #io_Ausgang_Ventil_10;	// (008)
      );
      =     #io_Ventil_in_Betrieb;
NETWORK
TITLE = Flankenauswertung Ausgang Ventil für Schalthäufigkeitzähler
//Es wird die Schalthäufigkeit der Ventile gezählt !  
      O     #io_Ausgang_Ventil_1;
      O     #io_Ausgang_Ventil_2;
      O     #io_Ausgang_Ventil_3;
      O     #io_Ausgang_Ventil_4;
      O     #io_Ausgang_Ventil_5;
      O     #io_Ausgang_Ventil_6;
      O     #io_Ausgang_Ventil_7;
      O     #io_Ausgang_Ventil_8;
      O     #io_Ausgang_Ventil_9;
      O     #io_Ausgang_Ventil_10;
      FP    DIX [AR2,P#32.3];	// Flankenmerker Ausgang (Struktur)
      =     #positive_Flanke;
NETWORK
TITLE = Schalthäufigkeitzähler
      ON    DIX [AR2,P#0.3];	// Kennung Schalthäufigkeitzähler ein (Struktur)
      ON    #positive_Flanke;
      JC    ESHZ;
      L     1.000000e+00;
      L     DID [AR2,P#34.0];	// Schalthäufigkeitzähler (Struktur)
      +R;
      T     DID [AR2,P#34.0];	// Schalthäufigkeitzähler (Struktur)
ESHZ: NOP   0;
NETWORK
TITLE = Schalthäufigkeitzähler zurücksetzten
      AN    DIX [AR2,P#32.0];	// Reset Schalthäufigkeitzähler (Struktur)
      JC    E_RS;
      L     0.000000e+00;
      T     DID [AR2,P#34.0];	// Schalthäufigkeitzähler (Struktur)
      CLR;
      =     DIX [AR2,P#32.0];	// Reset Schalthäufigkeitzähler (Struktur)
E_RS: NOP   0;
NETWORK
TITLE = Warnmeldung Schalthäufigkeitzähler erzeugen
      A(;
      L     DID [AR2,P#34.0];	// Schalthäufigkeitzähler (Struktur)
      L     DID [AR2,P#38.0];	// Sollwert Warnung (Struktur)
      >R;
      );
      A(;
      L     DID [AR2,P#38.0];	// Sollwert Warnung (Struktur)
      L     0.000000e+00;
      <>R;
      );
      =     DIX [AR2,P#32.1];	// Warnmeldung Schalthäufigkeitzähler (Struktur)
NETWORK
TITLE = Alarmmeldung Schalthäufigkeitzähler erzeugen
      A(;
      L     DID [AR2,P#34.0];	// Schalthäufigkeitzähler (Struktur)
      L     DID [AR2,P#42.0];	// Sollwert Alarm (Struktur)
      >R;
      );
      A(;
      L     DID [AR2,P#42.0];	// Sollwert Alarm (Struktur)
      L     0.000000e+00;
      <>R;
      );
      =     DIX [AR2,P#32.2];	// Warnmeldung Schalthäufigkeitzähler (Struktur)
NETWORK
TITLE = Objektstatus für Visualisation OP (011)(012)
//Stati:
//-------
//1 = kein Ventil angesteuert ==> Farbvorschlag weiß
//5 = ein ventil in Betrieb ==> Farbvorschlag grün
//
// 1 = nicht in Betrieb, keine Störung ==> Farbvorschlag grau
      L     1;
      AN    #io_Ventil_in_Betrieb;
      JC    disp;
// 5 = angesteuert, nicht in Betrieb, keine Störung ==> Farbvorschlag grün
      L     5;
      A     #io_Ventil_in_Betrieb;
      JC    disp;
      L     0;
disp: T     #Objektstatus;
NETWORK
TITLE = Daten in Struktur speichern
      A     #in_Anlage_ein;	// (014)
      =     DIX [AR2,P#5.5];	// (014) Anlage ein (Struktur)
      A     #io_Ausgang_Ventil_1;
      =     DIX [AR2,P#2.0];	// Ausgang Ventil 1 (Struktur)
      A     #io_Ausgang_Ventil_2;
      =     DIX [AR2,P#2.1];	// Ausgang Ventil 2 (Struktur)
      A     #io_Ausgang_Ventil_3;
      =     DIX [AR2,P#2.2];	// Ausgang Ventil 3 (Struktur)
      A     #io_Ausgang_Ventil_4;
      =     DIX [AR2,P#2.3];	// Ausgang Ventil 4 (Struktur)
      A     #io_Ausgang_Ventil_5;
      =     DIX [AR2,P#2.4];	// Ausgang Ventil 5 (Struktur)
      A     #io_Ausgang_Ventil_6;
      =     DIX [AR2,P#2.5];	// Ausgang Ventil 6 (Struktur)
      A     #io_Ausgang_Ventil_7;
      =     DIX [AR2,P#2.6];	// Ausgang Ventil 7 (Struktur)
      A     #io_Ausgang_Ventil_8;
      =     DIX [AR2,P#2.7];	// Ausgang Ventil 8 (Struktur)
      A     #io_Ausgang_Ventil_9;
      =     DIX [AR2,P#3.0];	// Ausgang Ventil 9 (Struktur)
      A     #io_Ausgang_Ventil_10;
      =     DIX [AR2,P#3.1];	// Ausgang Ventil 10 (Struktur)
      A     #io_Ventil_in_Betrieb;
      =     DIX [AR2,P#3.4];	// Ventil in Betrieb (Struktur)
      A     #Taktanzahl_erreicht;
      =     DIX [AR2,P#5.3];	// Taktanzahl erreicht (Struktur)
      L     #Zeitzaehler;
      T     DID [AR2,P#22.0];	// Impuls-/Pausezähler (Struktur)
      L     #Taktzaehler;
      T     DIW [AR2,P#28.0];	// Taktzähler (Struktur)
      L     #Objektstatus;	// (011)
      T     DIW [AR2,P#48.0];	// #Objektstatus  (Struktur)   // (011)
END_FUNCTION

FUNCTION "FC24 Binary-I Object" : VOID	// FC 24
TITLE = Block for debouncing and fault monitoring of a binary input
//Building:
//Date         Editor                                                     Version
//--------------------------------------------------------------------------------
//22.09.99     (jm)                                                       01.00.00
//
//Modifications:
//No. Date     Edit  Description                                    Index Version
//--------------------------------------------------------------------------------
//01  29.09.00 sra   komplette Überarbeitung / neue Struktur        ()    02.00.00
//02  16.06.05 sra   Änderung INC 1 -> + 1                         (002)  02.00.01
//03  04.09.06 sra   Änderung Störungsquittierung                  (003)  02.01.00
//04  08.07.10 jm    Störzeit 0 möglich                            (004)  02.01.01
//05  06.06.16 kal/sra komplette Überarbeitung (wie TIA-Portal)     ()    03.00.00
//06  12.06.16 sra   Änderung Signal "Eingang verarbeitet"         (006)  03.01.00
//
//________________________________________________________________________________
//Functional description:
//
//The Binary Input Object includes the following functions
//- The input can be turned (0 = input is active) -> configuration value
//- Depending on the Parameter "in_fault_state", it is possible to select whether
//  log. 0 or log. 1 will represent the fault.
//- The input signal can be debounced in both directions with a seperate time
//  -> Real values in structure
//- The input signal can be counted -> value in structure -> configuration value
//
//The main application for the function are level indicators.
//
VERSION : 0.0
VAR_INPUT
  in_Handbedienung_erlaubt : BOOL ;
  in_Anlage_ein : BOOL ;
  in_Eingang : BOOL ;
  in_Eingang_drehen : BOOL ;
  in_Eingang_entprellen : BOOL ;
  in_Stoerauswertung_aktiv : BOOL ;
  in_Quitt_Stoerung_noetig : BOOL ;
  in_Stoer_Zustand : BOOL ;
  in_Quitt_Stoerung : BOOL ;
END_VAR
VAR_IN_OUT
  io_Eingang_verarbeitet : BOOL ;
  io_Stoerung : BOOL ;
  io_Struktur : ANY ;
END_VAR
VAR_TEMP
  Eingang_nach_Drehung : BOOL ;
  Eingang_nach_Entprellung : BOOL ;
  Diskrepanz : BOOL ;
  Freigabe_Entprellung_HIG : BOOL ;
  Ausgang_Entprellung_HIGH : BOOL ;
  Freigabe_Entprellung_LOW : BOOL ;
  Ausgang_Entprellung_LOW : BOOL ;
  positive_Flanke : BOOL ;
  Objektstatus : INT ;
  Temp_DB : INT ;
  Sollzeit_Entprellung_HIG : REAL ;
  Istzeit_Entprellung_HIGH : REAL ;
  Sollzeit_Entprellung_LOW : REAL ;
  Istzeit_entprellung_LOW : REAL ;
END_VAR
BEGIN
NETWORK
TITLE = Anfangs-DW der Struktur aus ANY-Zeiger auslesen
      L     P##io_Struktur;
      LAR2;
      L     D [AR2,P#6.0];
      LAR2;
NETWORK
TITLE = Daten aus Struktur lesen
      A     DIX [AR2,P#3.4];
      =     #Eingang_nach_Drehung;
      A     DIX [AR2,P#3.5];
      =     #Eingang_nach_Entprellung;
      A     DIX [AR2,P#3.6];
      =     #Ausgang_Entprellung_HIGH;
      A     DIX [AR2,P#3.7];
      =     #Ausgang_Entprellung_LOW;
      L     DID [AR2,P#8.0];
      T     #Sollzeit_Entprellung_HIG;
      L     DID [AR2,P#12.0];
      T     #Istzeit_Entprellung_HIGH;
      L     DID [AR2,P#16.0];
      T     #Sollzeit_Entprellung_LOW;
      L     DID [AR2,P#20.0];
      T     #Istzeit_entprellung_LOW;
NETWORK
TITLE = Eingang ggf. drehen
      A     #in_Eingang;
      AN    #in_Eingang_drehen;
      O;
      AN    #in_Eingang;
      A     #in_Eingang_drehen;
      =     #Eingang_nach_Drehung;
NETWORK
TITLE = Umschaltung Hand-/Automatikmode 
      A     DIX [AR2,P#2.7];	// Handmode von Farbgrafik (Struktur)
      AN    DIX [AR2,P#3.1];	// Handmode gesperrt (Struktur)
      AN    "M 0.0 Lock Man.Operation";	// Handbedienung zentral sperren 
      S     DIX [AR2,P#2.6];	// Handmode zu Farbgrafik (Struktur)
      ON    DIX [AR2,P#2.7];	// Handmode von Farbgrafik (Struktur)
      ON    #in_Handbedienung_erlaubt;
      O     "M 0.0 Lock Man.Operation";	// Handbedienung zentral sperren 
      O     DIX [AR2,P#3.1];	// Handmode gesperrt (Struktur)
      R     DIX [AR2,P#2.6];	// Handmode zu Farbgrafik (Struktur)
      R     DIX [AR2,P#2.7];	// Handmode von Farbgrafik (Struktur)
NETWORK
TITLE = Handzustand im Automatikmode speichern
      AN    DIX [AR2,P#2.6];	// Handmode zu Farbgrafik (Struktur)
      JCN   SAM;
      A     #Eingang_nach_Drehung;
      AN    #in_Eingang_drehen;
      =     DIX [AR2,P#3.0];	// Zustand Handmode (Struktur)
      AN    #Eingang_nach_Drehung;
      A     #in_Eingang_drehen;
      =     DIX [AR2,P#3.0];	// Zustand Handmode (Struktur)
SAM:  NOP   0;
NETWORK
TITLE = Zustand nach Drehung im Handmode überschreiben
      A     DIX [AR2,P#2.6];	// Handmode zu Farbgrafik (Struktur)
      JCN   SHM;
      A     DIX [AR2,P#3.0];	// Zustand Handmode (Struktur)
      =     #Eingang_nach_Drehung;
SHM:  NOP   0;
NETWORK
TITLE = Diskrepanz feststellen
// Automode
      AN    DIX [AR2,P#2.6];	// Handmode zu Farbgrafik (Struktur)
      A     #in_Stoerauswertung_aktiv;
      AN    #in_Eingang;	//Störung = log. 0
      AN    #in_Stoer_Zustand;
      O;
      AN    DIX [AR2,P#2.6];	// Handmode zu Farbgrafik (Struktur)
      A     #in_Stoerauswertung_aktiv;
      A     #in_Eingang;	//Störung = log. 1
      A     #in_Stoer_Zustand;
      O;
// Handmode 
      A     DIX [AR2,P#2.6];	// Handmode zu Farbgrafik (Struktur)
      A     #in_Stoerauswertung_aktiv;
      AN    #Eingang_nach_Drehung;	//Störung = log. 0
      AN    #in_Stoer_Zustand;
      O;
      A     DIX [AR2,P#2.6];	// Handmode zu Farbgrafik (Struktur)
      A     #in_Stoerauswertung_aktiv;
      A     #Eingang_nach_Drehung;	//Störung = log. 1
      A     #in_Stoer_Zustand;
      =     #Diskrepanz;
NETWORK
TITLE = Stoerungszaehler
      A     #in_Quitt_Stoerung_noetig;
      AN    #in_Quitt_Stoerung;
      A     #io_Stoerung;
      O;
      A     #Diskrepanz;
      AN    #in_Quitt_Stoerung;
      O;
      AN    #in_Quitt_Stoerung_noetig;
      A     #Diskrepanz;
      JC    SZ1;
      L     0;	// Wenn keine Diskrepanz dann Zähler löschen
      T     DIW [AR2,P#6.0];	// Istzeit Störung (Struktur)
      JU    ESZ;
// Störungszähler in jeder Sekunde erhöhen
SZ1:  O     #io_Stoerung;
      ON    "M 4.5 Imp Cycle 1,0-sec";	// Sekundenimpuls (Standardmerker)
      JC    ESZ;
      L     DIW [AR2,P#6.0];	// Istzeit Störung (Struktur)
      +     1;	// (002)
      T     DIW [AR2,P#6.0];	// Istzeit Störung (Struktur)
ESZ:  NOP   0;
NETWORK
TITLE = Störmeldung ausgeben
      L     DIW [AR2,P#6.0];	// Istzeit Störung (Struktur)
      L     DIW [AR2,P#4.0];	// Sollzeit Störung (Struktur)
      >I;
      =     #io_Stoerung;
NETWORK
TITLE = Stoerung quittieren
      O     #Diskrepanz;	// Stoerung steht noch an
      ON    #io_Stoerung;
      JC    ESQ;
      ON    #in_Quitt_Stoerung_noetig;	// Stoerung muß quittiert werden ?
      JC    SQ1;	// Stoerung muß nicht quittiert werden
      A     #in_Quitt_Stoerung;
SQ1:  R     #io_Stoerung;
ESQ:  NOP   0;
NETWORK
TITLE = Entprellung HIGH
      A     #Eingang_nach_Drehung;
      A     #in_Eingang_entprellen;
      =     #Freigabe_Entprellung_HIG;
      CALL  "FC3 Cycle generator" (
           in_Freigabe              := #Freigabe_Entprellung_HIG,
           in_Reset                 := "M 0.3 Reset",
           in_Impuls                := "M 1.7 Cycle Timer-FC",
           in_Impulszeit_in_100ms   := "MW 6 Timer Val Cycle FCs",
           in_Verzoegerungsart      := B#16#45,
           in_Verzoegerungszeit     := #Sollzeit_Entprellung_HIG,
           io_Ausgangssignal        := #Ausgang_Entprellung_HIGH,
           io_Zeitzaehler           := #Istzeit_Entprellung_HIGH);
NETWORK
TITLE = Entprellung LOW
      AN    #Eingang_nach_Drehung;
      A     #in_Eingang_entprellen;
      =     #Freigabe_Entprellung_LOW;
      CALL  "FC3 Cycle generator" (
           in_Freigabe              := #Freigabe_Entprellung_LOW,
           in_Reset                 := "M 0.3 Reset",
           in_Impuls                := "M 1.7 Cycle Timer-FC",
           in_Impulszeit_in_100ms   := "MW 6 Timer Val Cycle FCs",
           in_Verzoegerungsart      := B#16#45,
           in_Verzoegerungszeit     := #Sollzeit_Entprellung_LOW,
           io_Ausgangssignal        := #Ausgang_Entprellung_LOW,
           io_Zeitzaehler           := #Istzeit_entprellung_LOW);
NETWORK
TITLE = Entprellung
      A     #Eingang_nach_Drehung;
      A     #in_Eingang_entprellen;
      A     #Ausgang_Entprellung_HIGH;
      S     #Eingang_nach_Entprellung;
      AN    #Eingang_nach_Drehung;
      A     #in_Eingang_entprellen;
      A     #Ausgang_Entprellung_LOW;
      R     #Eingang_nach_Entprellung;
      NOP   0;
NETWORK
TITLE = verarbeitetes Eingangssignal zuweisen
// Automatikmode
      AN    DIX [AR2,P#2.6];	// Handmode zu Farbgrafik (Struktur)
      AN    #in_Eingang_entprellen;
      A     #Eingang_nach_Drehung;
      AN    #io_Stoerung;	// (006)
      O;
// Automatikmode
      AN    DIX [AR2,P#2.6];	// Handmode zu Farbgrafik (Struktur)
      A     #in_Eingang_entprellen;
      A     #Eingang_nach_Entprellung;
      AN    #io_Stoerung;	// (006)
      O;
// Handmode 
      A     DIX [AR2,P#2.6];	// Handmode zu Farbgrafik (Struktur)
      A     DIX [AR2,P#3.0];	// Zustand Handmode (Struktur)
      AN    #in_Eingang_drehen;
      AN    #io_Stoerung;	// (006)
      O;
// Handmode 
      A     DIX [AR2,P#2.6];	// Handmode zu Farbgrafik (Struktur)
      AN    DIX [AR2,P#3.0];	// Zustand Handmode (Struktur)
      A     #in_Eingang_drehen;
      AN    #io_Stoerung;	// (006)
      =     #io_Eingang_verarbeitet;
NETWORK
TITLE = Flankenauswertung Ausgang Ventil für Schalthäufigkeitzähler
      A     #io_Eingang_verarbeitet;
      FP    DIX [AR2,P#24.3];	// Flankenmerker Ausgang (Struktur)
      =     #positive_Flanke;
NETWORK
TITLE = Schalthäufigkeitzähler
      ON    DIX [AR2,P#0.3];	// Kennung Schalthäufigkeitzähler ein (Struktur)
      ON    #positive_Flanke;
      JC    ESHZ;
      L     1.000000e+00;
      L     DID [AR2,P#26.0];	// Schalthäufigkeitzähler (Struktur)
      +R;
      T     DID [AR2,P#26.0];	// Schalthäufigkeitzähler (Struktur)
ESHZ: NOP   0;
NETWORK
TITLE = Schalthäufigkeitzähler zurücksetzten
      AN    DIX [AR2,P#24.0];	// Reset Schalthäufigkeitzähler (Struktur)
      JC    E_RS;
      L     0.000000e+00;
      T     DID [AR2,P#26.0];	// Schalthäufigkeitzähler (Struktur)
      CLR;
      =     DIX [AR2,P#24.0];	// Reset Schalthäufigkeitzähler (Struktur)
E_RS: NOP   0;
NETWORK
TITLE = Warnmeldung Schalthäufigkeitszähler erzeugen
      A(;
      L     DID [AR2,P#26.0];	// Schalthäufigkeitzähler (Struktur)
      L     DID [AR2,P#30.0];	// Sollwert Warnung (Struktur)
      >R;
      );
      A(;
      L     DID [AR2,P#30.0];	// Sollwert Warnung (Struktur)
      L     0.000000e+00;
      <>R;
      );
      =     DIX [AR2,P#24.1];	// Warnmeldung Schalthäufigkeitzähler (Struktur)
NETWORK
TITLE = Alarmmeldung Schalthäufigkeitszähler erzeugen
      A(;
      L     DID [AR2,P#26.0];	// Schalthäufigkeitzähler (Struktur)
      L     DID [AR2,P#34.0];	// Sollwert Alarm (Struktur)
      >R;
      );
      A(;
      L     DID [AR2,P#34.0];	// Sollwert Alarm (Struktur)
      L     0.000000e+00;
      <>R;
      );
      =     DIX [AR2,P#24.2];	// Alarmmeldung Schalthäufigkeitzähler (Struktur)
NETWORK
TITLE = Objektstatus für Visualisation OP (009) (010)
// 19 = Anlage nicht ein (interlock) ==> Farbvorschlag orange
      L     19;
      AN    #in_Anlage_ein;
      AN    #io_Stoerung;
      JC    disp;
// 1 = nicht betaetigt
      L     1;
      AN    #io_Eingang_verarbeitet;
      AN    #io_Stoerung;
      AN    DIX [AR2,P#1.0];	// Kennung "invers"
      O;
      A     #io_Eingang_verarbeitet;
      AN    #io_Stoerung;
      A     DIX [AR2,P#1.0];	// Kennung "invers"
      JC    disp;
// 5 = betätigt
      L     5;
      A     #io_Eingang_verarbeitet;
      AN    #io_Stoerung;
      AN    DIX [AR2,P#1.0];	// Kennung "invers"
      O;
      AN    #io_Eingang_verarbeitet;
      AN    #io_Stoerung;
      A     DIX [AR2,P#1.0];	// Kennung "invers"
      JC    disp;
// 16 = Störung
      L     16;
      A     #io_Stoerung;
      JC    disp;
      L     0;
disp: T     #Objektstatus;
NETWORK
TITLE = Daten in Struktur kopieren
      A     #io_Eingang_verarbeitet;
      =     DIX [AR2,P#2.0];	// Eingang verarbeitet (Struktur)
      A     #in_Eingang;
      =     DIX [AR2,P#2.1];	// Eingang (Struktur)
      A     #in_Eingang_drehen;
      =     DIX [AR2,P#2.2];	// Eingang drehen (Struktur)
      A     #in_Eingang_entprellen;
      =     DIX [AR2,P#2.3];	// Eingang entprellen (Struktur)
      A     #in_Stoer_Zustand;
      =     DIX [AR2,P#2.4];	// Störzustand (Struktur)
      A     #io_Stoerung;
      =     DIX [AR2,P#2.5];	// Störung (Struktur)
      A     #in_Anlage_ein;	// (006)
      =     DIX [AR2,P#3.2];	// (006) Anlage ein (Struktur) 
      A     #Eingang_nach_Drehung;
      =     DIX [AR2,P#3.4];
      A     #Eingang_nach_Entprellung;
      =     DIX [AR2,P#3.5];
      A     #Ausgang_Entprellung_HIGH;
      =     DIX [AR2,P#3.6];
      A     #Ausgang_Entprellung_LOW;
      =     DIX [AR2,P#3.7];
      AN    #Ausgang_Entprellung_HIGH;
      JCN   noHi;
      L     #Istzeit_Entprellung_HIGH;
      T     DID [AR2,P#12.0];
noHi: NOP   0;
      AN    #Ausgang_Entprellung_LOW;
      JCN   noLo;
      L     #Istzeit_entprellung_LOW;
      T     DID [AR2,P#20.0];
noLo: NOP   0;
      L     #Objektstatus;
      T     DIW [AR2,P#48.0];	// #Objektstatus  (Struktur) 
END_FUNCTION

FUNCTION "FC30 Pre -assign DB" : VOID	// FC 30
TITLE = Baustein vorbelegen
//Erstellung:
//Datum        Bearbeiter                                                 Version
//--------------------------------------------------------------------------------
//08.12.98     R.Schaffert (sra)                                          01.00.00
//
//Änderungen:
//Nr. Datum    Bearb Beschreibung                                   Marke Version
//--------------------------------------------------------------------------------
//01  13.04.00 sra   Fehlerbehebung (1 Byte zuviel belegt)                01.00.01
//02  25.08.00 sra   Fehlerbehebung Zeigerberechnung                      01.00.02
//
//________________________________________________________________________________
//Beschreibung:
//
//Diese Funktion beschreibt die angegebenen Worte eines Datenbausteins mit dem im 
//Parameter "Wert" eingetragenen Wert.
//
AUTHOR : sra
FAMILY : AZO
VERSION : 0.0
VAR_INPUT
  DB_Nr : INT ;	//Datenbausteinnummer
  DW_Anfang : INT ;	//Anfangs-Datenwort im Datenbaustein
  Anzahl_Bytes : INT ;	//Anzahl der Bytes die vorbelegt werden sollen
  Wert : INT ;	//Wert mit dem der Bereich vorbelegt werden soll
END_VAR
VAR_TEMP
  Datenbaustein : INT ;
  Ptr_aktuelles_Datenbyte : DWORD ;
  Ptr_Ende_Datenbyte : DWORD ;
END_VAR
BEGIN
NETWORK
TITLE = Anzahl Worte prüfen
      L     #Anzahl_Bytes;
      L     0;
      <=I;
      JC    Ende;
NETWORK
TITLE = Datenbaustein öffnen
      L     #DB_Nr;
      T     #Datenbaustein;
      OPN   DB [#Datenbaustein];
NETWORK
TITLE = Pointer belegen
      L     #DW_Anfang;
      SLD   3;
      T     #Ptr_aktuelles_Datenbyte;
      L     #Anzahl_Bytes;
      L     #DW_Anfang;
      +I;
      SLD   3;
      T     #Ptr_Ende_Datenbyte;
NETWORK
TITLE = Wert schreiben
Loop: NOP   0;
      L     #Wert;
      T     DBB [#Ptr_aktuelles_Datenbyte];
      L     #Ptr_aktuelles_Datenbyte;	// Wortadresse um 1 erhöhen
      L     P#1.0;
      +D;
      T     #Ptr_aktuelles_Datenbyte;
      L     #Ptr_Ende_Datenbyte;
      <D;
      JC    Loop;
Ende: NOP   0;
END_FUNCTION

FUNCTION "FC40 copy Obj-IF Master" : VOID	// FC 40
TITLE = SST an Slave
//Erstellung:
//Datum        Bearbeiter                                                 Version
//--------------------------------------------------------------------------------
//22.03.01     R.Schaffert (sra)                                          01.00.00
//
//Änderungen:
//Nr. Datum    Bearb Beschreibung                                   Marke Version
//--------------------------------------------------------------------------------
//01  16.08.01 sra   Fehlerbeseitigung  Daten löschen               (001) 01.00.01
//02  31.08.01 sra   Daten von Ziel auch löschen wenn Ziel-DB 0 ist (002) 01.00.02
//
//________________________________________________________________________________
//Beschreibung: 
//
//Der Baustein kopiert die Schnittstelle, die durch den ANY-Zeiger festgelegt 
//ist, 
//an einen "Slave". Sobald ein Bit in der Steuerbitleiste gesetzt ist reagiert 
//der 
//Slave und antwortet. Ist kein Bit in der Steuerbitleiste belegt, baut der Slave 
//die Schnittstelle ab und kann durch anderen Master belegt werden.
//!!Die Steuerbitleiste ist immer das letzte Wort in der Schnittstelle!!
//
//Anwendung z.B. bei Kommunikation mehrere Waage <-> mehrere Silo  
// 
//
AUTHOR : sra
FAMILY : AZO
VERSION : 0.0
VAR_INPUT
  i_Freigabe : BOOL ;	//Freigabe der Kopierfunktion
  i_Ziel_DB : INT ;	//Ziel-Datenbaustein
  i_Ziel_DW : INT ;	//Ziel-Datenwort im Ziel-Datenbaustein
  i_SST_von_Ziel : ANY ;	//ANY-Zeiger auf Schnittstellen von Slave
  i_SST_an_Ziel : ANY ;	//ANY-Zeiger auf Schnittstellen an Slave
END_VAR
VAR_OUTPUT
  Ziel_frei : BOOL ;	//"Slave" ist nicht durch anderen Master belegt,die Daten können umkopiert werden
END_VAR
VAR_TEMP
  Quell_DB : INT ;
  SST_an_Anfangs_DW : INT ;
  SST_an_Laenge : INT ;
  SST_von_Anfangs_DW : INT ;
  SST_von_Laenge : INT ;
  Ziel_DB : INT ;
  Zaehler : INT ;
  Fehler_Blockkopieren : INT ;
END_VAR
BEGIN
NETWORK
TITLE = ANY Zeiger "SST_von_Ziel" zerlegen
      L     P##i_SST_von_Ziel;
      LAR2;
      L     W [AR2,P#2.0];
      T     #SST_von_Laenge;
      L     D [AR2,P#6.0];
      L     DW#16#FFFFFF;
      AD;
      SRD   3;
      T     #SST_von_Anfangs_DW;
NETWORK
TITLE = ANY Zeiger "SST_an_Ziel" zerlegen
      L     P##i_SST_an_Ziel;
      LAR2;
      L     W [AR2,P#2.0];
      T     #SST_an_Laenge;
      L     W [AR2,P#4.0];
      T     #Quell_DB;
      L     D [AR2,P#6.0];
      L     DW#16#FFFFFF;
      AD;
      SRD   3;
      T     #SST_an_Anfangs_DW;
NETWORK
TITLE = Prüfen ob Ziel-DB <> 0
      L     #i_Ziel_DB;
      L     0;
      ==I;
      JC    DEL1;	// 002
NETWORK
TITLE = Prüfen ob Slave belegt ist
      L     #i_Ziel_DB;
      T     #Ziel_DB;
      OPN   DB [#Ziel_DB];
      L     #i_Ziel_DW;
      SLD   3;
      LAR2;
      O(;	// Slave bereits belegt ?
      L     DBW [AR2,P#0.0];
      L     #Quell_DB;
      ==I;
      );
      O(;	// Slave frei ?
      L     DBW [AR2,P#0.0];
      L     0;
      ==I;
      );
      =     #Ziel_frei;
NETWORK
TITLE = Daten von Ziel löschen
DEL1: OPN   DB [#Quell_DB];
      L     #SST_von_Anfangs_DW;
      SLD   3;
      LAR2;
      L     #SST_von_Laenge;
DEL2: T     #Zaehler;
      L     0;
      T     DBB [AR2,P#0.0];
      L     P#1.0;	// (001)
      +AR2;	// (001)
      L     #Zaehler;
      LOOP  DEL2;
      ON    #i_Freigabe;
      ON    #Ziel_frei;
      O(;	// (002)
      L     #i_Ziel_DB;	// (002)
      L     0;	// (002)
      ==I;	// (002)
      );	// (002)
      BEC;
NETWORK
TITLE = Daten an Slave kopieren
      L     #SST_an_Anfangs_DW;
      SLD   3;
      LAR2;
      L     #Quell_DB;
      T     DBW [AR2,P#0.0];
      L     #SST_von_Anfangs_DW;
      T     DBW [AR2,P#2.0];
      CALL  "FC5 Block Transfer" (
           Quell_Typ                := B#16#44,
           Quell_DB                 := #Quell_DB,
           Quell_DW                 := #SST_an_Anfangs_DW,
           Ziel_Typ                 := B#16#44,
           Ziel_DB                  := #i_Ziel_DB,
           Ziel_DW                  := #i_Ziel_DW,
           Block_Laenge             := #SST_an_Laenge,
           outFehler                := #Fehler_Blockkopieren);
END_FUNCTION

FUNCTION "FC41 copy Obj-IF Slave" : VOID	// FC 41
TITLE = SST an Master
//Erstellung:
//Datum        Bearbeiter                                                 Version
//--------------------------------------------------------------------------------
//22.03.01     R.Schaffert (sra)                                          01.00.00
//
//Änderungen:
//Nr. Datum    Bearb Beschreibung                                   Marke Version
//--------------------------------------------------------------------------------
//01  00.00.00 xxx   xxx                                            ???   01.xx.xx
//
//________________________________________________________________________________
//Beschreibung: 
//
//Der Baustein kopiert die Schnittstelle, die durch den ANY-Zeiger festgelegt 
//ist, an einen "Master". Sobald ein Bit in der Steuerbitleiste gesetzt ist 
//reagiert der Slave und antwortet. Ist kein Bit in der Steuerbitleiste belegt, 
//baut der Slave die Schnittstelle ab und kann durch anderen Master belegt werden.
//!!Die Steuerbitleiste ist immer das letzte Wort in der Schnittstelle!!
//
//Anwendung z.B. bei Kommunikation mehrere Waage <-> mehrere Silo  
// 
//
//
AUTHOR : sra
FAMILY : AZO
VERSION : 0.0
VAR_INPUT
  i_SST_von_Ziel : ANY ;	//ANY-Zeiger auf Schnittstelle von Master
  i_SST_an_Ziel : ANY ;	//ANY-Zeiger auf Schnittstelle an Master
END_VAR
VAR_TEMP
  SST_an_Anfangs_DW : INT ;
  SST_an_Laenge : INT ;
  SST_von_Anfangs_DW : INT ;
  SST_von_Laenge : INT ;
  Ptr_SST_von_Anfangs_DW : DWORD ;
  Ptr_SST_von_Steuerbits : DWORD ;	//Steuerbits = Anfangs-DW + Länge -2
  Quell_DB : INT ;
  Ziel_DB : INT ;
  Ziel_DW : INT ;
  Fehler_Blockkopieren : INT ;
END_VAR
BEGIN
NETWORK
TITLE = ANY Zeiger "SST_von_Ziel" zerlegen
      L     P##i_SST_von_Ziel;
      LAR2;
      L     W [AR2,P#2.0];	// Länge der Struktur
      T     #SST_von_Laenge;
      L     D [AR2,P#6.0];	// Anfangs-DW der Struktur
      L     DW#16#FFFFFF;
      AD;
      SRD   3;
      T     #SST_von_Anfangs_DW;
NETWORK
TITLE = ANY Zeiger "SST_an_Ziel" zerlegen
      L     P##i_SST_an_Ziel;
      LAR2;
      L     W [AR2,P#2.0];
      T     #SST_an_Laenge;
      L     W [AR2,P#4.0];
      T     #Quell_DB;
      L     D [AR2,P#6.0];
      L     DW#16#FFFFFF;
      AD;
      SRD   3;
      T     #SST_an_Anfangs_DW;
NETWORK
TITLE = Pointer bilden
      L     #SST_von_Anfangs_DW;
      SLD   3;
      T     #Ptr_SST_von_Anfangs_DW;
      L     #SST_von_Anfangs_DW;
      L     #SST_von_Laenge;
      +I;
      L     2;
      -I;
      SLD   3;
      T     #Ptr_SST_von_Steuerbits;
NETWORK
TITLE = Prüfen ob Anforderung vorhanden
      OPN   DB [#Quell_DB];
      O(;
      L     DBW [#Ptr_SST_von_Anfangs_DW];	// Ziel-DB
      L     0;
      ==I;
      );
      O(;
      L     DBW [#Ptr_SST_von_Steuerbits];	// Steuerbits
      L     0;
      ==I;
      );
      JC    DEL;
NETWORK
TITLE = Daten an Master kopieren
      LAR2  #Ptr_SST_von_Anfangs_DW;
      L     DBW [AR2,P#0.0];	// Ziel-DB aus Struktur "SST_von" ermitteln
      T     #Ziel_DB;
      L     DBW [AR2,P#2.0];	// Ziel-DW aus Struktur "SST_von" ermitteln
      T     #Ziel_DW;
      CALL  "FC5 Block Transfer" (
           Quell_Typ                := B#16#44,
           Quell_DB                 := #Quell_DB,
           Quell_DW                 := #SST_an_Anfangs_DW,
           Ziel_Typ                 := B#16#44,
           Ziel_DB                  := #Ziel_DB,
           Ziel_DW                  := #Ziel_DW,
           Block_Laenge             := #SST_an_Laenge,
           outFehler                := #Fehler_Blockkopieren);
NETWORK
TITLE = Daten von Master löschen
DEL:  L     DBW [#Ptr_SST_von_Steuerbits];
      L     0;
      <>I;
      JC    DELS;
      L     0;
      T     DBW [#Ptr_SST_von_Anfangs_DW];
DELS: L     0;
      T     DBW [#Ptr_SST_von_Steuerbits];
END_FUNCTION

DATA_BLOCK "DB2 Simulation"	// DB 2
VERSION : 0.0
"FB2 Simulation"
BEGIN
END_DATA_BLOCK

DATA_BLOCK "DB3 global Info"	// DB 3
AUTHOR : sra
FAMILY : AZO
VERSION : 0.0
  STRUCT
   OB1_Info : STRUCT
    OB1_DATE_TIME : DATE_AND_TIME ;	//Date and time OB1 started
    OB1_PREV_CYCLE : INT ;	//Cycle time of previous OB1 scan (milliseconds)
    OB1_MIN_CYCLE : INT ;	//Minimum cycle time of OB1 (milliseconds)
    OB1_MAX_CYCLE : INT ;	//Maximum cycle time of OB1 (milliseconds)
    reserve : ARRAY  [0 .. 14 ] OF BYTE ;
   END_STRUCT ;
   Fehler_OB_Info : STRUCT
    Zeitfehler_OB80 : BOOL ;	//Zeitfehler OB 80
    Stromversorgung_OB81 : BOOL ;	//Stromversorgungsfehler OB 81
    Diagnose_Alarm_OB82 : BOOL ;	//Diagnose-Alarm OB82
    Ziehen_Stecken_OB83 : BOOL ;	//Ziehen/Stecken-Alarm OB83
    CPU_Hardware_OB84 : BOOL ;	//CPU-Hardwarefehler OB84
    Programmablauf_OB85 : BOOL ;	//Programmablauffehler OB85
    Baugr_tr_ausfall_OB86 : BOOL ;	//Baugruppenträgerausfall OB86
    Kommunikation_OB87 : BOOL ;	//Kommunikationsfehler OB87
    Programmierfehler_OB121 : BOOL ;	//Programmierfehler OB121
    Periphzugriff_OB122 : BOOL ;	//Peripheriezugriffsfehler OB 122
    Bearbeitungsabbruch_OB88 : BOOL ;	//Bearbeitungsabbruch eines Bausteins OB88
    Battery_fault : BOOL ;	//Battery fault with SFC51
    reserve_word : WORD ;
    OB_80_Fault_ID : BYTE ;	//Fehlercode OB 80
    OB_81_Fault_ID : BYTE ;	//Fehlercode OB 81
    OB_82_Fault_ID : BYTE ;	//Fehlercode OB 82
    OB_83_Fault_ID : BYTE ;	//Fehlercode OB 83
    OB_84_Fault_ID : BYTE ;	//Fehlercode OB 84
    OB_85_Fault_ID : BYTE ;	//Fehlercode OB 85
    OB_86_Fault_ID : BYTE ;	//Fehlercode OB 86
    OB_87_Fault_ID : BYTE ;	//Fehlercode OB 87
    OB_121_Fault_ID : BYTE ;	//Fehlercode OB 121
    OB_122_Fault_ID : BYTE ;	//Fehlercode OB 122
    OB_88_Fault_ID : BYTE ;	//Fehlercode OB 122
    reserve : ARRAY  [16 .. 29 ] OF BYTE ;
   END_STRUCT ;
   RDSYSST : STRUCT
    BUSY : BOOL ;
    RETVAL : INT ;
    SLZ_HEADER : STRUCT
     LENTHDR : WORD ;
     N_DR : WORD ;
    END_STRUCT ;
    DR : STRUCT
     Data_1 : BYTE ;
     Data_2 : BYTE ;
     Data_3 : BYTE ;
     Data_4 : BYTE ;
     Data_5 : BYTE ;
     Data_6 : BYTE ;
     Data_7 : BYTE ;
     Data_8 : BYTE ;
     Data_9 : BYTE ;
     Data_10 : BYTE ;
     Data_11 : BYTE ;
     Data_12 : BYTE ;
     Data_13 : BYTE ;
     Data_14 : BYTE ;
     Data_15 : BYTE ;
     Data_16 : BYTE ;
     Data_17 : BYTE ;
     Data_18 : BYTE ;
     Data_19 : BYTE ;
     Data_20 : BYTE ;
    END_STRUCT ;
   END_STRUCT ;
  END_STRUCT ;	
BEGIN
END_DATA_BLOCK

DATA_BLOCK "DB30 Daten from/to SCADA"	// DB 30
AUTHOR : sra
FAMILY : hsh
VERSION : 0.0
"FB30 Daten from/to SCADA"
BEGIN
END_DATA_BLOCK

DATA_BLOCK "DB32 Inputs"	// DB 32
AUTHOR : sra
FAMILY : SCADA
VERSION : 0.0
"FB32 Inputs to SCADA"
BEGIN
END_DATA_BLOCK

DATA_BLOCK "DV33 Outputs"	// DB 33
AUTHOR : sra
FAMILY : SCADA
VERSION : 0.0
"FB33 Outputs to SCADA"
BEGIN
END_DATA_BLOCK

DATA_BLOCK "DB34 Faults"	// DB 34
AUTHOR : sra
FAMILY : AZO
VERSION : 0.0
"FB34 Fault evaluation"
BEGIN
END_DATA_BLOCK

DATA_BLOCK "DB35 Acknowledge Faults"	// DB 35
VERSION : 0.1
  STRUCT
   Quittierung : ARRAY  [0 .. 1023, 0 .. 7 ] OF BOOL  := FALSE;
   Quittierung_Spiegelungen : ARRAY  [0 .. 1023, 0 .. 7 ] OF BOOL  := FALSE;
  END_STRUCT ;	
BEGIN
END_DATA_BLOCK

DATA_BLOCK "PRODUCTION_DB"	// DB 1000
VERSION : 0.0
"PRODUCTION"
BEGIN
END_DATA_BLOCK

DATA_BLOCK "HOPPER_HP01_DB"	// DB 1001
AUTHOR : ilia
VERSION : 0.0
"HOPPER"
BEGIN
END_DATA_BLOCK

DATA_BLOCK "HOPPER_HP02_DB"	// DB 1002
AUTHOR : ilia
VERSION : 0.0
"HOPPER"
BEGIN
END_DATA_BLOCK

DATA_BLOCK "REC01_DB"	// DB 1011
AUTHOR : ilia
VERSION : 0.0
"REC01"
BEGIN
END_DATA_BLOCK

DATA_BLOCK "PMP01_DB"	// DB 1051
VERSION : 0.0
"PMP01"
BEGIN
END_DATA_BLOCK

DATA_BLOCK "FC01_RV_HOPPERS_DB"	// DB 10001
VERSION : 0.0
"FC01_RV_HOPPERS"
BEGIN
END_DATA_BLOCK

ORGANIZATION_BLOCK "OB1 Cycle"	// OB 1
TITLE = "Main Program Sweep (Cycle)"
//Creation:
//Date:            Author:                                               Version
//--------------------------------------------------------------------------------
//14.04.2017      Ilia Bedniakov(ilia)                                   01.00.00
//
//Changes:
//No. Date:        Who       Description                           Mark   Version 
//--------------------------------------------------------------------------------
//01
//________________________________________________________________________________
//Function:
VERSION : 0.1
VAR_TEMP
  OB1_EV_CLASS : BYTE ;	//Bits 0-3 = 1 (Coming event), Bits 4-7 = 1 (Event class 1)
  OB1_SCAN_1 : BYTE ;	//1 (Cold restart scan 1 of OB 1), 3 (Scan 2-n of OB 1)
  OB1_PRIORITY : BYTE ;	//Priority of OB Execution
  OB1_OB_NUMBR : BYTE ;	//1 (Organization block 1, OB1)
  OB1_RESERVED_1 : BYTE ;	//Reserved for system
  OB1_RESERVED_2 : BYTE ;	//Reserved for system
  OB1_PREV_CYCLE : INT ;	//Cycle time of previous OB1 scan (milliseconds)
  OB1_MIN_CYCLE : INT ;	//Minimum cycle time of OB1 (milliseconds)
  OB1_MAX_CYCLE : INT ;	//Maximum cycle time of OB1 (milliseconds)
  OB1_DATE_TIME : DATE_AND_TIME ;	//Date and time OB1 started
  DUMMY_INT : INT ;
  dummy_bool : BOOL ;
END_VAR
BEGIN
NETWORK
TITLE = Simunation
      CLR;
//    SET   
      =     "M 0.5 InternalSimulation";
      A     "M 0.5 InternalSimulation";
      JCN   NS;	// No simulation
      CALL  "FB2 Simulation" , "DB2 Simulation";
NS:   NOP   0;
NETWORK
TITLE = Datum, Uhrzeit und Zykluszeiten in DB3 kopieren
      CALL  "SFC 20 BLKMOV" (
           SRCBLK                   := #OB1_DATE_TIME,
           RET_VAL                  := #DUMMY_INT,
           DSTBLK                   := "DB3 global Info".OB1_Info.OB1_DATE_TIME);
      L     #OB1_PREV_CYCLE;
      T     "DB3 global Info".OB1_Info.OB1_PREV_CYCLE;
      L     #OB1_MIN_CYCLE;
      T     "DB3 global Info".OB1_Info.OB1_MIN_CYCLE;
      L     #OB1_MAX_CYCLE;
      T     "DB3 global Info".OB1_Info.OB1_MAX_CYCLE;
NETWORK
TITLE = Standardsignale
      CALL  "FC13 Standard Signals" (
           in_E_Sicherung_OK        := "ES_03_01_602",
           in_Basistakt_Timer       := "M 4.1 Imp Cycle 0,2-sec",
           in_Zeit_Basistakt_100ms  := 2,
           o_Lampe_Stoer_Sicherung  := #dummy_bool,
           o_Stoerung_Sicherung     := DB34.DBX 5.7);
NETWORK
TITLE = data from / to VISU
      CALL  "FB30 Daten from/to SCADA" , "DB30 Daten from/to SCADA";
      CALL  "FB32 Inputs to SCADA" , "DB32 Inputs";
      CALL  "FB33 Outputs to SCADA" , "DV33 Outputs";
NETWORK
TITLE = fault evaluation
      CALL  "FB34 Fault evaluation" , "DB34 Faults";
NETWORK
TITLE = Production Line
      CALL  "PRODUCTION" , "PRODUCTION_DB";
END_ORGANIZATION_BLOCK

ORGANIZATION_BLOCK "OB 80 Zeitfehler-OB"	// OB 80
TITLE = Zeitfehler
//Erstellung:
//Datum        Bearbeiter                                                 Version
//--------------------------------------------------------------------------------
//03.06.98     Rainer Schaffert (sra)                                     01.00.00
//
//Änderungen:
//Nr. Datum    Bearb Beschreibung                                   Marke Version
//--------------------------------------------------------------------------------
//01  
//
//________________________________________________________________________________
//OB wird bei Zeitfehler bearbeitet
//
AUTHOR : sra
FAMILY : error_OB
NAME : time_err
VERSION : 0.1
VAR_TEMP
  OB80_EV_CLASS : BYTE ;	//16#35, Event class 3, Entering event state, Internal fault event
  OB80_FLT_ID : BYTE ;	//16#XX, Fault identifcation code
  OB80_PRIORITY : BYTE ;	//26 (Priority of 1 is lowest)
  OB80_OB_NUMBR : BYTE ;	//80 (Organization block 80, OB80)
  OB80_RESERVED_1 : BYTE ;	//Reserved for system
  OB80_RESERVED_2 : BYTE ;	//Reserved for system
  OB80_ERROR_INFO : WORD ;	//Error information on event
  OB80_ERR_EV_CLASS : BYTE ;	//Class of event causing error
  OB80_ERR_EV_NUM : BYTE ;	//Number of event causing error
  OB80_OB_PRIORITY : BYTE ;	//Priority of OB causing error
  OB80_OB_NUM : BYTE ;	//Number of OB causing error
  OB80_DATE_TIME : DATE_AND_TIME ;	//Date and time OB80 started
END_VAR
BEGIN
NETWORK
TITLE = Fehlermeldung erzeugen
//Fehlermeldung erzeugen
//
//Fehlercode B#16#01 : Zykluszeit überschritten
//                     OB80_ERROR_INFO: Laufzeit des letzten Zyklus
//           
//           B#16#02 : Der angeforderte OB ist noch in Bearbeitung
//
//           B#16#07 : Überlauf des OB-Anforderungspuffers für die aktuelle 
//                     Prioritätsklasse
//
//           B#16#05 : abgelaufener Urzeitalarm durch Urzeitsprung
//
//           B#16#06 : abgelaufener Urzeitalarm bei Wiedereintritt 
//
      L     #OB80_FLT_ID;
      L     B#16#0;
      <>I;
      =     "DB3 global Info".Fehler_OB_Info.Zeitfehler_OB80;
      L     #OB80_FLT_ID;
      T     "DB3 global Info".Fehler_OB_Info.OB_80_Fault_ID;
END_ORGANIZATION_BLOCK

ORGANIZATION_BLOCK "OB 82 Diagnosealarm-OB"	// OB 82
TITLE = Diagnose-Alarm
//Erstellung:
//Datum        Bearbeiter                                                 Version
//--------------------------------------------------------------------------------
//03.06.98     Rainer Schaffert (sra)                                     01.00.00
//
//Änderungen:
//Nr. Datum    Bearb Beschreibung                                   Marke Version
//--------------------------------------------------------------------------------
//01  
//
//________________________________________________________________________________
//OB wird bei Diagnose-Alarm bearbeitet
//
AUTHOR : sra
FAMILY : error_OB
NAME : diagn_OB
VERSION : 0.1
VAR_TEMP
  OB82_EV_CLASS : BYTE ;	//16#39, Event class 3, Entering event state, Internal fault event
  OB82_FLT_ID : BYTE ;	//16#XX, Fault identifcation code
  OB82_PRIORITY : BYTE ;	//26/28 (Priority of 1 is lowest)
  OB82_OB_NUMBR : BYTE ;	//82 (Organization block 82, OB82)
  OB82_RESERVED_1 : BYTE ;	//Reserved for system
  OB82_IO_FLAG : BYTE ;	//Input (01010100), Output (01010101)
  OB82_MDL_ADDR : INT ;	//Base address of module with fault
  OB82_MDL_DEFECT : BOOL ;	//Module defective
  OB82_INT_FAULT : BOOL ;	//Internal fault
  OB82_EXT_FAULT : BOOL ;	//External fault
  OB82_PNT_INFO : BOOL ;	//Point information
  OB82_EXT_VOLTAGE : BOOL ;	//External voltage low
  OB82_FLD_CONNCTR : BOOL ;	//Field wiring connector missing
  OB82_NO_CONFIG : BOOL ;	//Module has no configuration data
  OB82_CONFIG_ERR : BOOL ;	//Module has configuration error
  OB82_MDL_TYPE : BYTE ;	//Type of module
  OB82_SUB_NDL_ERR : BOOL ;	//Sub-Module is missing or has error
  OB82_COMM_FAULT : BOOL ;	//Communication fault
  OB82_MDL_STOP : BOOL ;	//Module is stopped
  OB82_WTCH_DOG_FLT : BOOL ;	//Watch dog timer stopped module
  OB82_INT_PS_FLT : BOOL ;	//Internal power supply fault
  OB82_PRIM_BATT_FLT : BOOL ;	//Primary battery is in fault
  OB82_BCKUP_BATT_FLT : BOOL ;	//Backup battery is in fault
  OB82_RESERVED_2 : BOOL ;	//Reserved for system
  OB82_RACK_FLT : BOOL ;	//Rack fault, only for bus interface module
  OB82_PROC_FLT : BOOL ;	//Processor fault
  OB82_EPROM_FLT : BOOL ;	//EPROM fault
  OB82_RAM_FLT : BOOL ;	//RAM fault
  OB82_ADU_FLT : BOOL ;	//ADU fault
  OB82_FUSE_FLT : BOOL ;	//Fuse fault
  OB82_HW_INTR_FLT : BOOL ;	//Hardware interupt input in fault
  OB82_RESERVED_3 : BOOL ;	//Reserved for system
  OB82_DATE_TIME : DATE_AND_TIME ;	//Date and time OB82 started
END_VAR
BEGIN
NETWORK
TITLE = Fehlermeldung erzeugen
//Fehlermeldung erzeugen
//
//Fehlercode B#16#42 : 
//
      A(;
      L     #OB82_EV_CLASS;
      L     B#16#39;	// kommendes Ereignis
      ==I;
      );
      A(;
      L     #OB82_FLT_ID;
      L     B#16#0;
      <>I;
      );
      =     "DB3 global Info".Fehler_OB_Info.Diagnose_Alarm_OB82;
      L     #OB82_FLT_ID;
      T     "DB3 global Info".Fehler_OB_Info.OB_82_Fault_ID;
END_ORGANIZATION_BLOCK

ORGANIZATION_BLOCK "OB 83 Ziehen-/Stecken-OB"	// OB 83
TITLE = Ziehen/Stecken-Alarm
//Erstellung:
//Datum        Bearbeiter                                                 Version
//--------------------------------------------------------------------------------
//03.06.98     Rainer Schaffert (sra)                                     01.00.00
//
//Änderungen:
//Nr. Datum    Bearb Beschreibung                                   Marke Version
//--------------------------------------------------------------------------------
//01  
//
//________________________________________________________________________________
//OB wird bei Ziehen/Stecken-Alarm bearbeitet
//
AUTHOR : sra
FAMILY : AZO
VERSION : 0.0
VAR_TEMP
  OB83_EV_CLASS : BYTE ;	//16#38/39, Event class 3, module inserted/removed (8/9)
  OB83_FLT_ID : BYTE ;	//16#XX, Fault identifcation code
  OB83_PRIORITY : BYTE ;	//26/28 (Priority of 1 is lowest)
  OB83_OB_NUMBR : BYTE ;	//83 (Organization block 83, OB83)
  OB83_RESERVED_1 : BYTE ;	//Reserved for system
  OB83_MDL_ID : BYTE ;	//Input module (01010100), Output module (01010101)
  OB83_MDL_ADDR : WORD ;	//Base address of module with point fault
  OB83_RACK_NUM : WORD ;	//Number of rack that has module with point fault
  OB83_MDL_TYPE : WORD ;	//Module type with point fault
  OB83_DATE_TIME : DATE_AND_TIME ;	//Date and time OB83 started
END_VAR
BEGIN
NETWORK
TITLE = Fehlermeldung erzeugen
//Fehlermeldung erzeugen
//
//Fehlercode B#16#61 : Baugruppe gezogen bzw. nicht ansprechbar (bei 
//                     Ereignisklasse B#16#39)
//                     Baugruppe gesteckt, Baugruppentyp ok (bei
//                     Ereignisklasse B#16#38)
//           
//           B#16#63 : Baugruppe gesteckt, jedoch falscher Baugruppentyp
//
//           B#16#64 : Baugruppe gesteckt, jedoch gestört(Typkennung nicht lesbar)
//
      A(;
      L     #OB83_EV_CLASS;
      L     B#16#39;	// kommendes Ereignis
      ==I;
      );
      A(;
      L     #OB83_FLT_ID;
      L     B#16#0;
      <>I;
      );
      =     "DB3 global Info".Fehler_OB_Info.Ziehen_Stecken_OB83;
      L     #OB83_FLT_ID;
      T     "DB3 global Info".Fehler_OB_Info.OB_83_Fault_ID;
END_ORGANIZATION_BLOCK

ORGANIZATION_BLOCK "OB 85 Prgablauffehler-OB"	// OB 85
TITLE = Programmablauffehler
//Erstellung:
//Datum        Bearbeiter                                                 Version
//--------------------------------------------------------------------------------
//03.06.98     Rainer Schaffert (sra)                                     01.00.00
//
//Änderungen:
//Nr. Datum    Bearb Beschreibung                                   Marke Version
//--------------------------------------------------------------------------------
//01  
//
//________________________________________________________________________________
//OB wird bei Programmablauffehler bearbeitet
//
//
AUTHOR : sra
FAMILY : AZO
VERSION : 0.0
VAR_TEMP
  OB85_EV_CLASS : BYTE ;	//16#35 Event class 3
  OB85_FLT_ID : BYTE ;	//16#XX, Fault identification code
  OB85_PRIORITY : BYTE ;	//26 (Priority of 1 is lowest)
  OB85_OB_NUMBR : BYTE ;	//85 (Organization block 85, OB85)
  OB85_RESERVED_1 : BYTE ;	//Reserved for system
  OB85_RESERVED_2 : BYTE ;	//Reserved for system
  OB85_RESERVED_3 : INT ;	//Reserved for system
  OB85_ERR_EV_CLASS : BYTE ;	//Class of event causing error
  OB85_ERR_EV_NUM : BYTE ;	//Number of event causing error
  OB85_OB_PRIOR : BYTE ;	//Priority of OB causing error
  OB85_OB_NUM : BYTE ;	//Number of OB causing error
  OB85_DATE_TIME : DATE_AND_TIME ;	//Date and time OB85 started
END_VAR
BEGIN
NETWORK
TITLE = Fehlermeldung erzeugen
//Fehlermeldung erzeugen
//
//Fehlercode B#16#A1 : Das Programm oder das Betriebssystem erzeugt ein 
//                     Startereignis für einen OB, der nicht in die CPU geladen 
//                     ist.
//
//           B#16#A2 : Das Programm oder das Betriebssystem erzeugt ein 
//                     Startereignis für einen OB, der nicht in die CPU geladen 
//                     ist.
//
//           B#16#A3 : Fehler beim Zugriff des Betriebssystems auf einen Baustein
//
//           B#16#B1 : Peripheriezugriffsfehler beim Aktualisieren des 
//                     Gesamtprozessabbildes der Eingänge
//
//           B#16#B1 : Peripheriezugriffsfehler beim Aktualisieren des            
//                     Gesamtprozessabbildes der Ausgänge
//
      L     #OB85_FLT_ID;
      L     B#16#0;
      <>I;
      =     "DB3 global Info".Fehler_OB_Info.Programmablauf_OB85;
      L     #OB85_FLT_ID;
      T     "DB3 global Info".Fehler_OB_Info.OB_85_Fault_ID;
END_ORGANIZATION_BLOCK

ORGANIZATION_BLOCK "OB 86 Baugr träger-OB"	// OB 86
TITLE = Baugruppenträgerausfall
//Erstellung:
//Datum        Bearbeiter                                                 Version
//--------------------------------------------------------------------------------
//03.06.98     Rainer Schaffert (sra)                                     01.00.00
//
//Änderungen:
//Nr. Datum    Bearb Beschreibung                                   Marke Version
//--------------------------------------------------------------------------------
//01  
//
//________________________________________________________________________________
//OB wird bei Baugruppenträgerausfall bearbeitet
//
AUTHOR : sra
FAMILY : AZO
VERSION : 0.0
VAR_TEMP
  OB86_EV_CLASS : BYTE ;	//16#38/39 Event class 3
  OB86_FLT_ID : BYTE ;	//16#C1/C4/C5, Fault identification code
  OB86_PRIORITY : BYTE ;	//26/28 (Priority of 1 is lowest)
  OB86_OB_NUMBR : BYTE ;	//86 (Organization block 86, OB86)
  OB86_RESERVED_1 : BYTE ;	//Reserved for system
  OB86_RESERVED_2 : BYTE ;	//Reserved for system
  OB86_MDL_ADDR : WORD ;	//Depending on fault identification code
  OB86_RACKS_FLTD : ARRAY  [0 .. 31 ] OF BOOL ;	//Racks in fault
  OB86_DATE_TIME : DATE_AND_TIME ;	//Date and time OB86 started
END_VAR
BEGIN
NETWORK
TITLE = Fehlermeldung erzeugen
//Fehlermeldung erzeugen
//
//Fehlercode B#16#C1 : Baugruppenträgerausfall
//
//           B#16#C2 : Baugruppenträgerwiederkehr (Baugruppenträgerausfall gehend 
//                     mit Abweichung Soll-/Istausbau)
//
//           B#16#C3 : Dezentrale Peripherie: Ausfall eines DP-Mastersystems
//
//           B#16#C4 : Ausfall einer DP-Station
//
//           B#16#C5 : Störung einer DP-Station
//
      A(;
      L     #OB86_EV_CLASS;
      L     B#16#39;	// kommendes Ereignis
      ==I;
      );
      A(;
      L     #OB86_FLT_ID;
      L     B#16#0;
      <>I;
      );
      =     "DB3 global Info".Fehler_OB_Info.Baugr_tr_ausfall_OB86;
      L     #OB86_FLT_ID;
      T     "DB3 global Info".Fehler_OB_Info.OB_86_Fault_ID;
END_ORGANIZATION_BLOCK

ORGANIZATION_BLOCK "OB 87 Kommunikations-OB"	// OB 87
TITLE = Kommunikationsfehler
//Erstellung:
//Datum        Bearbeiter                                                 Version
//--------------------------------------------------------------------------------
//03.06.98     Rainer Schaffert (sra)                                     01.00.00
//
//Änderungen:
//Nr. Datum    Bearb Beschreibung                                   Marke Version
//--------------------------------------------------------------------------------
//01  
//
//________________________________________________________________________________
//OB wird bei Kommunikationsfehler bearbeitet
//
AUTHOR : sra
FAMILY : AZO
VERSION : 0.0
VAR_TEMP
  OB87_EV_CLASS : BYTE ;	//16#35 Event class 3
  OB87_FLT_ID : BYTE ;	//16#XX, Fault identifcation code
  OB87_PRIORITY : BYTE ;	//26 (Priority of 1 is lowest)
  OB87_OB_NUMBR : BYTE ;	//87 (Organization block 87, OB87)
  OB87_RESERVED_1 : BYTE ;	//Reserved for system
  OB87_RESERVED_2 : BYTE ;	//Reserved for system
  OB87_RESERVED_3 : WORD ;	//Reserved for system
  OB87_RESERVED_4 : DWORD ;	//Reserved for system
  OB87_DATE_TIME : DATE_AND_TIME ;	//Date and time OB87 started
END_VAR
BEGIN
NETWORK
TITLE = Fehlermeldung erzeugen
//Fehlermeldung erzeugen
//
//Fehlercode B#16#D2 : Senden der Diagnoseeinträge nicht möglich
//
//           B#16#D3 : Synchronisationsdiagramme können nicht gesendet werden
//
//           B#16#D4 : Unzulässiger Uhrzeitsprung durch Uhrzeitsynchronisation
//
//           B#16#D5 : Fehler bei Übernahme der Synchronisationszeit
//
//           B#16#E1 : Falsche Telegrammkennung bei Globaldatenkommunikation
//
//           B#16#E3 : Telegrammlängenfehler bei Globaldatenkommunikation
//
//           B#16#E4 : Unzulässige GD-Paketnummer empfangen
//
//           B#16#E2 : GD-Paketstatus ist nicht in einen DP-eintragbar
//
//           B#16#E5 : Fehler bei Zugriff auf DB beim Datenaustausch über 
//                     Kommunikationsfunktionsbausteine
//
//           B#16#E6 : GD-Gesamtstatus ist nicht in DB eintragbar
//
      L     #OB87_FLT_ID;
      L     B#16#0;
      <>I;
      =     "DB3 global Info".Fehler_OB_Info.Kommunikation_OB87;
      L     #OB87_FLT_ID;
      T     "DB3 global Info".Fehler_OB_Info.OB_87_Fault_ID;
END_ORGANIZATION_BLOCK

ORGANIZATION_BLOCK "OB 100 Neustart-OB"	// OB 100
TITLE = Neustart
//Erstellung:
//Datum        Bearbeiter                                                 Version
//--------------------------------------------------------------------------------
//04.09.2001   R.Schaffert (sra)                                          01.00.00
//  
//Änderungen:
//Nr. Datum    Bearb Änderung                                       Marke  Version
//--------------------------------------------------------------------------------
//
//________________________________________________________________________________
//Programm wird am Anfang von OB 1 fortgesetzt
AUTHOR : sra
FAMILY : AZO
VERSION : 0.0
VAR_TEMP
  OB100_EV_CLASS : BYTE ;	//16#13, Event class 1, Entering event state, Event logged in diagnostic buffer
  OB100_STRTUP : BYTE ;	//16#81/82/83/84 Method of startup
  OB100_PRIORITY : BYTE ;	//27 (Priority of 1 is lowest)
  OB100_OB_NUMBR : BYTE ;	//100 (Organization block 100, OB100)
  OB100_RESERVED_1 : BYTE ;	//Reserved for system
  OB100_RESERVED_2 : BYTE ;	//Reserved for system
  OB100_STOP : WORD ;	//Event that caused CPU to stop (16#4xxx)
  OB100_STRT_INFO : DWORD ;	//Information on how system started
  OB100_DATE_TIME : DATE_AND_TIME ;	//Date and time OB100 started
END_VAR
BEGIN
NETWORK
TITLE = Neustartmerker setzen
      SET;
      S     "M 1.3 Hot/WarmRestartPLC";
END_ORGANIZATION_BLOCK

